LIN {X 0,Y 229.65,Z 466.167,A -85,B 0,C 180,E1 -20819.777,E2 -20819.777} C_VEL
LIN {X 0,Y 225.789,Z 455.718,A -85,B 0,C 180,E1 -20821.607,E2 -20821.607} C_VEL
LIN {X 0,Y 220.787,Z 444.949,A -85,B 0,C 180,E1 -20823.43,E2 -20823.43} C_VEL
LIN {X 0,Y 215.475,Z 435.139,A -85,B 0,C 180,E1 -20825.063,E2 -20825.063} C_VEL
LIN {X 0,Y 214,Z 432.562,A -85,B 0,C 180,E1 -20825.471,E2 -20825.471} C_VEL
LIN {X 0,Y 213.743,Z 431.361,A -85,B 0,C 180,E1 -20825.592,E2 -20825.592} C_VEL
LIN {X 0,Y 213.779,Z 431.357,A -85,B 0,C 180,E1 -20828.655,E2 -20828.655} C_VEL
LIN {X 0,Y 213.791,Z 431.354,A -85,B 0,C 180,E1 -20831.107,E2 -20831.107} C_VEL
LIN {X 0,Y 213.806,Z 431.352,A -85,B 0,C 180,E1 -20833.686,E2 -20833.686} C_VEL
LIN {X 0,Y 213.727,Z 431.361,A -85,B 0,C 180,E1 -20838.88,E2 -20838.88} C_VEL
LIN {X 0,Y 213.75,Z 431.36,A -85,B 0,C 180,E1 -20843.714,E2 -20843.714} C_VEL
LIN {X 0,Y 213.794,Z 431.352,A -85,B 0,C 180,E1 -20848.725,E2 -20848.725} C_VEL
LIN {X 0,Y 213.824,Z 431.35,A -85,B 0,C 180,E1 -20852.604,E2 -20852.604} C_VEL
LIN {X 0,Y 213.85,Z 431.346,A -85,B 0,C 180,E1 -20856.954,E2 -20856.954} C_VEL
LIN {X 0,Y 213.942,Z 431.334,A -85,B 0,C 180,E1 -20862.805,E2 -20862.805} C_VEL
LIN {X 0,Y 213.979,Z 431.329,A -85,B 0,C 180,E1 -20866.709,E2 -20866.709} C_VEL
LIN {X 0,Y 214.166,Z 431.302,A -85,B 0,C 180,E1 -20870.557,E2 -20870.557} C_VEL
LIN {X 0,Y 214.226,Z 431.299,A -85,B 0,C 180,E1 -20872.461,E2 -20872.461} C_VEL
LIN {X 0,Y 214.445,Z 431.245,A -85,B 0,C 180,E1 -20878.123,E2 -20878.123} C_VEL
LIN {X 0,Y 214.549,Z 431.244,A -85,B 0,C 180,E1 -20880.001,E2 -20880.001} C_VEL
LIN {X 0,Y 214.445,Z 431.271,A -85,B 0,C 180,E1 -20881.879,E2 -20881.879} C_VEL
LIN {X 0,Y 214.248,Z 431.3,A -85,B 0,C 180,E1 -20887.541,E2 -20887.541} C_VEL
LIN {X 0,Y 214.042,Z 431.325,A -85,B 0,C 180,E1 -20891.363,E2 -20891.363} C_VEL
LIN {X 0,Y 213.934,Z 431.338,A -85,B 0,C 180,E1 -20895.238,E2 -20895.238} C_VEL
LIN {X 0,Y 213.841,Z 431.349,A -85,B 0,C 180,E1 -20899.188,E2 -20899.188} C_VEL
LIN {X 0,Y 213.848,Z 431.35,A -85,B 0,C 180,E1 -20903.228,E2 -20903.228} C_VEL
LIN {X 0,Y 213.864,Z 431.711,A -85,B 0,C 180,E1 -20907.393,E2 -20907.393} C_VEL
LIN {X 0,Y 214.059,Z 433.405,A -85,B 0,C 180,E1 -20911.691,E2 -20911.691} C_VEL
LIN {X 0,Y 214.301,Z 435.41,A -85,B 0,C 180,E1 -20916.18,E2 -20916.18} C_VEL
LIN {X 0,Y 214.681,Z 437.889,A -85,B 0,C 180,E1 -20921.154,E2 -20921.154} C_VEL
LIN {X 0,Y 214.855,Z 439.419,A -85,B 0,C 180,E1 -20923.976,E2 -20923.976} C_VEL
LIN {X 0,Y 214.881,Z 440.961,A -85,B 0,C 180,E1 -20926.62,E2 -20926.62} C_VEL
LIN {X 0,Y 214.731,Z 442.501,A -85,B 0,C 180,E1 -20929.112,E2 -20929.112} C_VEL
LIN {X 0,Y 213.923,Z 445.534,A -85,B 0,C 180,E1 -20933.747,E2 -20933.747} C_VEL
LIN {X 0,Y 213.756,Z 446.179,A -85,B 0,C 180,E1 -20934.654,E2 -20934.654} C_VEL
LIN {X 0,Y 214.719,Z 449.544,A -85,B 0,C 180,E1 -20935.029,E2 -20935.029} C_VEL
LIN {X 0,Y 218.657,Z 461.683,A -85,B 0,C 180,E1 -20936.689,E2 -20936.689} C_VEL
LIN {X 0,Y 221.392,Z 472.962,A -85,B 0,C 180,E1 -20938.374,E2 -20938.374} C_VEL
LIN {X 0,Y 222.956,Z 483.058,A -85,B 0,C 180,E1 -20939.999,E2 -20939.999} C_VEL
LIN {X 0,Y 223.803,Z 491.807,A -85,B 0,C 180,E1 -20941.557,E2 -20941.557} C_VEL
LIN {X 0,Y 223.936,Z 501.293,A -85,B 0,C 180,E1 -20943.435,E2 -20943.435} C_VEL
LIN {X 0,Y 223.732,Z 505.859,A -85,B 0,C 180,E1 -20944.41,E2 -20944.41} C_VEL
LIN {X 0,Y 220.785,Z 516.308,A -85,B 0,C 180,E1 -20946.818,E2 -20946.818} C_VEL
LIN {X 0,Y 219.001,Z 523.013,A -85,B 0,C 180,E1 -20948.742,E2 -20948.742} C_VEL
LIN {X 0,Y 216.849,Z 529.814,A -85,B 0,C 180,E1 -20951.089,E2 -20951.089} C_VEL
LIN {X 0,Y 215.381,Z 534.744,A -85,B 0,C 180,E1 -20953.138,E2 -20953.138} C_VEL
LIN {X 0,Y 213.858,Z 537.614,A -85,B 0,C 180,E1 -20954.475,E2 -20954.475} C_VEL
LIN {X 0,Y 209.85,Z 541.622,A -85,B 0,C 180,E1 -20956.666,E2 -20956.666} C_VEL
LIN {X 0,Y 206.092,Z 545.045,A -85,B 0,C 180,E1 -20959.012,E2 -20959.012} C_VEL
LIN {X 0,Y 204.987,Z 546.698,A -85,B 0,C 180,E1 -20960.564,E2 -20960.564} C_VEL
LIN {X 0,Y 204.442,Z 549.502,A -85,B 0,C 180,E1 -20964.08,E2 -20964.08} C_VEL
LIN {X 0,Y 204.339,Z 550.566,A -85,B 0,C 180,E1 -20966.055,E2 -20966.055} C_VEL
LIN {X 0,Y 204.365,Z 551.161,A -85,B 0,C 180,E1 -20968.029,E2 -20968.029} C_VEL
LIN {X 0,Y 204.429,Z 551.319,A -85,B 0,C 180,E1 -20970,E2 -20970} C_VEL
LIN {X 0,Y 204.365,Z 551.161,A -85,B 0,C 180,E1 -20971.97,E2 -20971.97} C_VEL
LIN {X 0,Y 204.36,Z 550.491,A -85,B 0,C 180,E1 -20974.184,E2 -20974.184} C_VEL
LIN {X 0,Y 204.675,Z 548.109,A -85,B 0,C 180,E1 -20977.894,E2 -20977.894} C_VEL
LIN {X 0,Y 205.363,Z 545.153,A -85,B 0,C 180,E1 -20980.849,E2 -20980.849} C_VEL
LIN {X 0,Y 206.414,Z 541.157,A -85,B 0,C 180,E1 -20983.788,E2 -20983.788} C_VEL
LIN {X 0,Y 208.046,Z 536.024,A -85,B 0,C 180,E1 -20986.686,E2 -20986.686} C_VEL
LIN {X 0,Y 209.722,Z 530.759,A -85,B 0,C 180,E1 -20989.07,E2 -20989.07} C_VEL
LIN {X 0,Y 211.844,Z 524.444,A -85,B 0,C 180,E1 -20991.402,E2 -20991.402} C_VEL
LIN {X 0,Y 213.537,Z 518.486,A -85,B 0,C 180,E1 -20993.262,E2 -20993.262} C_VEL
LIN {X 0,Y 215.597,Z 511.56,A -85,B 0,C 180,E1 -20995.072,E2 -20995.072} C_VEL
LIN {X 0,Y 217.256,Z 505.648,A -85,B 0,C 180,E1 -20996.409,E2 -20996.409} C_VEL
LIN {X 0,Y 217.344,Z 495.828,A -85,B 0,C 180,E1 -20998.546,E2 -20998.546} C_VEL
LIN {X 0,Y 216.761,Z 486.56,A -85,B 0,C 180,E1 -21000.341,E2 -21000.341} C_VEL
LIN {X 0,Y 215.486,Z 477.1,A -85,B 0,C 180,E1 -21002.006,E2 -21002.006} C_VEL
LIN {X 0,Y 213.303,Z 466.615,A -85,B 0,C 180,E1 -21003.699,E2 -21003.699} C_VEL
LIN {X 0,Y 210.591,Z 457.078,A -85,B 0,C 180,E1 -21005.148,E2 -21005.148} C_VEL
LIN {X 0,Y 207.683,Z 448.976,A -85,B 0,C 180,E1 -21006.358,E2 -21006.358} C_VEL
LIN {X 0,Y 206.901,Z 445.966,A -85,B 0,C 180,E1 -21006.726,E2 -21006.726} C_VEL
LIN {X 0,Y 207.477,Z 443.775,A -85,B 0,C 180,E1 -21010.059,E2 -21010.059} C_VEL
LIN {X 0,Y 207.749,Z 442.248,A -85,B 0,C 180,E1 -21012.576,E2 -21012.576} C_VEL
LIN {X 0,Y 207.813,Z 440.729,A -85,B 0,C 180,E1 -21015.25,E2 -21015.25} C_VEL
LIN {X 0,Y 207.522,Z 438.25,A -85,B 0,C 180,E1 -21019.948,E2 -21019.948} C_VEL
LIN {X 0,Y 207.228,Z 435.972,A -85,B 0,C 180,E1 -21024.791,E2 -21024.791} C_VEL
LIN {X 0,Y 206.982,Z 434.053,A -85,B 0,C 180,E1 -21029.38,E2 -21029.38} C_VEL
LIN {X 0,Y 206.751,Z 432.425,A -85,B 0,C 180,E1 -21033.774,E2 -21033.774} C_VEL
LIN {X 0,Y 206.756,Z 432.236,A -85,B 0,C 180,E1 -21038.042,E2 -21038.042} C_VEL
LIN {X 0,Y 206.871,Z 432.219,A -85,B 0,C 180,E1 -21042.195,E2 -21042.195} C_VEL
LIN {X 0,Y 206.893,Z 432.214,A -85,B 0,C 180,E1 -21046.243,E2 -21046.243} C_VEL
LIN {X 0,Y 207.13,Z 432.185,A -85,B 0,C 180,E1 -21050.231,E2 -21050.231} C_VEL
LIN {X 0,Y 207.185,Z 432.178,A -85,B 0,C 180,E1 -21052.201,E2 -21052.201} C_VEL
LIN {X 0,Y 207.379,Z 432.152,A -85,B 0,C 180,E1 -21058.057,E2 -21058.057} C_VEL
LIN {X 0,Y 207.511,Z 432.119,A -85,B 0,C 180,E1 -21059.999,E2 -21059.999} C_VEL
LIN {X 0,Y 207.378,Z 432.124,A -85,B 0,C 180,E1 -21061.941,E2 -21061.941} C_VEL
LIN {X 0,Y 207.164,Z 432.18,A -85,B 0,C 180,E1 -21067.798,E2 -21067.798} C_VEL
LIN {X 0,Y 206.977,Z 432.202,A -85,B 0,C 180,E1 -21071.754,E2 -21071.754} C_VEL
LIN {X 0,Y 206.862,Z 432.211,A -85,B 0,C 180,E1 -21075.77,E2 -21075.77} C_VEL
LIN {X 0,Y 206.779,Z 432.222,A -85,B 0,C 180,E1 -21079.868,E2 -21079.868} C_VEL
LIN {X 0,Y 206.758,Z 432.225,A -85,B 0,C 180,E1 -21084.071,E2 -21084.071} C_VEL
LIN {X 0,Y 206.739,Z 432.231,A -85,B 0,C 180,E1 -21088.418,E2 -21088.418} C_VEL
LIN {X 0,Y 206.704,Z 432.236,A -85,B 0,C 180,E1 -21092.955,E2 -21092.955} C_VEL
LIN {X 0,Y 206.721,Z 432.235,A -85,B 0,C 180,E1 -21097.73,E2 -21097.73} C_VEL
LIN {X 0,Y 206.744,Z 432.233,A -85,B 0,C 180,E1 -21101.596,E2 -21101.596} C_VEL
LIN {X 0,Y 206.741,Z 432.232,A -85,B 0,C 180,E1 -21105.55,E2 -21105.55} C_VEL
LIN {X 0,Y 206.739,Z 432.232,A -85,B 0,C 180,E1 -21109.768,E2 -21109.768} C_VEL
LIN {X 0,Y 206.711,Z 432.331,A -85,B 0,C 180,E1 -21113.059,E2 -21113.059} C_VEL
LIN {X 0,Y 207.683,Z 435.05,A -85,B 0,C 180,E1 -21113.417,E2 -21113.417} C_VEL
LIN {X 0,Y 209.172,Z 437.265,A -85,B 0,C 180,E1 -21113.847,E2 -21113.847} C_VEL
LIN {X 0,Y 214.507,Z 447.106,A -85,B 0,C 180,E1 -21115.615,E2 -21115.615} C_VEL
LIN {X 0,Y 218.684,Z 456.158,A -85,B 0,C 180,E1 -21117.262,E2 -21117.262} C_VEL
LIN {X 0,Y 222.353,Z 465.597,A -85,B 0,C 180,E1 -21119.035,E2 -21119.035} C_VEL
LIN {X 0,Y 225.766,Z 476.018,A -85,B 0,C 180,E1 -21121.121,E2 -21121.121} C_VEL
LIN {X 0,Y 229.479,Z 484.805,A -85,B 0,C 180,E1 -21123.22,E2 -21123.22} C_VEL
LIN {X 0,Y 234.862,Z 494.211,A -85,B 0,C 180,E1 -21125.874,E2 -21125.874} C_VEL
LIN {X 0,Y 241.471,Z 502.648,A -85,B 0,C 180,E1 -21128.645,E2 -21128.645} C_VEL
LIN {X 0,Y 249.05,Z 510.339,A -85,B 0,C 180,E1 -21131.527,E2 -21131.527} C_VEL
LIN {X 0,Y 256.368,Z 516.421,A -85,B 0,C 180,E1 -21134.09,E2 -21134.09} C_VEL
LIN {X 0,Y 263.767,Z 521.712,A -85,B 0,C 180,E1 -21136.585,E2 -21136.585} C_VEL
LIN {X 0,Y 270.068,Z 525.746,A -85,B 0,C 180,E1 -21138.71,E2 -21138.71} C_VEL
LIN {X 0,Y 277.243,Z 530.01,A -85,B 0,C 180,E1 -21141.347,E2 -21141.347} C_VEL
LIN {X 0,Y 280.836,Z 531.995,A -85,B 0,C 180,E1 -21142.812,E2 -21142.812} C_VEL
LIN {X 0,Y 283.81,Z 533.702,A -85,B 0,C 180,E1 -21144.316,E2 -21144.316} C_VEL
LIN {X 0,Y 285.973,Z 535.014,A -85,B 0,C 180,E1 -21145.772,E2 -21145.772} C_VEL
LIN {X 0,Y 288.419,Z 536.106,A -85,B 0,C 180,E1 -21147.495,E2 -21147.495} C_VEL
LIN {X 0,Y 289.599,Z 536.494,A -85,B 0,C 180,E1 -21148.61,E2 -21148.61} C_VEL
LIN {X 0,Y 290.596,Z 536.662,A -85,B 0,C 180,E1 -21150,E2 -21150} C_VEL
LIN {X 0,Y 289.595,Z 536.494,A -85,B 0,C 180,E1 -21151.391,E2 -21151.391} C_VEL
LIN {X 0,Y 287.975,Z 535.95,A -85,B 0,C 180,E1 -21152.798,E2 -21152.798} C_VEL
LIN {X 0,Y 285.954,Z 535.014,A -85,B 0,C 180,E1 -21154.229,E2 -21154.229} C_VEL
LIN {X 0,Y 282.8,Z 533.095,A -85,B 0,C 180,E1 -21156.257,E2 -21156.257} C_VEL
LIN {X 0,Y 280.804,Z 531.995,A -85,B 0,C 180,E1 -21157.189,E2 -21157.189} C_VEL
LIN {X 0,Y 274.892,Z 528.624,A -85,B 0,C 180,E1 -21159.566,E2 -21159.566} C_VEL
LIN {X 0,Y 267.715,Z 524.214,A -85,B 0,C 180,E1 -21162.123,E2 -21162.123} C_VEL
LIN {X 0,Y 258.513,Z 518.022,A -85,B 0,C 180,E1 -21165.186,E2 -21165.186} C_VEL
LIN {X 0,Y 250.424,Z 511.545,A -85,B 0,C 180,E1 -21167.981,E2 -21167.981} C_VEL
LIN {X 0,Y 242.862,Z 504.195,A -85,B 0,C 180,E1 -21170.799,E2 -21170.799} C_VEL
LIN {X 0,Y 235.936,Z 495.724,A -85,B 0,C 180,E1 -21173.66,E2 -21173.66} C_VEL
LIN {X 0,Y 230.601,Z 487.089,A -85,B 0,C 180,E1 -21176.18,E2 -21176.18} C_VEL
LIN {X 0,Y 226.199,Z 477.235,A -85,B 0,C 180,E1 -21178.617,E2 -21178.617} C_VEL
LIN {X 0,Y 222.351,Z 465.618,A -85,B 0,C 180,E1 -21180.963,E2 -21180.963} C_VEL
LIN {X 0,Y 219.408,Z 457.77,A -85,B 0,C 180,E1 -21182.441,E2 -21182.441} C_VEL
LIN {X 0,Y 214.209,Z 446.412,A -85,B 0,C 180,E1 -21184.497,E2 -21184.497} C_VEL
LIN {X 0,Y 208.574,Z 436.22,A -85,B 0,C 180,E1 -21186.355,E2 -21186.355} C_VEL
LIN {X 0,Y 207.02,Z 433.644,A -85,B 0,C 180,E1 -21186.817,E2 -21186.817} C_VEL
LIN {X 0,Y 206.702,Z 432.238,A -85,B 0,C 180,E1 -21187.013,E2 -21187.013} C_VEL
LIN {X 0,Y 206.721,Z 432.235,A -85,B 0,C 180,E1 -21191.589,E2 -21191.589} C_VEL
LIN {X 0,Y 206.671,Z 432.24,A -85,B 0,C 180,E1 -21195.571,E2 -21195.571} C_VEL
LIN {X 0,Y 206.67,Z 432.24,A -85,B 0,C 180,E1 -21199.753,E2 -21199.753} C_VEL
LIN {X 0,Y 206.729,Z 432.234,A -85,B 0,C 180,E1 -21204.696,E2 -21204.696} C_VEL
LIN {X 0,Y 206.721,Z 432.233,A -85,B 0,C 180,E1 -21209.34,E2 -21209.34} C_VEL
LIN {X 0,Y 206.73,Z 432.231,A -85,B 0,C 180,E1 -21213.773,E2 -21213.773} C_VEL
LIN {X 0,Y 206.756,Z 432.23,A -85,B 0,C 180,E1 -21218.044,E2 -21218.044} C_VEL
LIN {X 0,Y 206.872,Z 432.217,A -85,B 0,C 180,E1 -21222.198,E2 -21222.198} C_VEL
LIN {X 0,Y 206.912,Z 432.209,A -85,B 0,C 180,E1 -21226.247,E2 -21226.247} C_VEL
LIN {X 0,Y 207.104,Z 432.181,A -85,B 0,C 180,E1 -21230.232,E2 -21230.232} C_VEL
LIN {X 0,Y 207.167,Z 432.18,A -85,B 0,C 180,E1 -21232.202,E2 -21232.202} C_VEL
LIN {X 0,Y 207.381,Z 432.123,A -85,B 0,C 180,E1 -21238.059,E2 -21238.059} C_VEL
LIN {X 0,Y 207.514,Z 432.119,A -85,B 0,C 180,E1 -21240.001,E2 -21240.001} C_VEL
LIN {X 0,Y 207.382,Z 432.151,A -85,B 0,C 180,E1 -21241.943,E2 -21241.943} C_VEL
LIN {X 0,Y 207.188,Z 432.178,A -85,B 0,C 180,E1 -21247.799,E2 -21247.799} C_VEL
LIN {X 0,Y 206.975,Z 432.205,A -85,B 0,C 180,E1 -21251.757,E2 -21251.757} C_VEL
LIN {X 0,Y 206.867,Z 432.217,A -85,B 0,C 180,E1 -21255.772,E2 -21255.772} C_VEL
LIN {X 0,Y 206.785,Z 432.228,A -85,B 0,C 180,E1 -21259.87,E2 -21259.87} C_VEL
LIN {X 0,Y 206.765,Z 432.231,A -85,B 0,C 180,E1 -21264.073,E2 -21264.073} C_VEL
LIN {X 0,Y 206.753,Z 432.419,A -85,B 0,C 180,E1 -21266.226,E2 -21266.226} C_VEL
LIN {X 0,Y 206.983,Z 434.052,A -85,B 0,C 180,E1 -21270.62,E2 -21270.62} C_VEL
LIN {X 0,Y 207.24,Z 436.124,A -85,B 0,C 180,E1 -21275.522,E2 -21275.522} C_VEL
LIN {X 0,Y 207.532,Z 438.281,A -85,B 0,C 180,E1 -21280.049,E2 -21280.049} C_VEL
LIN {X 0,Y 207.816,Z 440.733,A -85,B 0,C 180,E1 -21284.75,E2 -21284.75} C_VEL
LIN {X 0,Y 207.713,Z 442.682,A -85,B 0,C 180,E1 -21288.107,E2 -21288.107} C_VEL
LIN {X 0,Y 207.079,Z 445.313,A -85,B 0,C 180,E1 -21292.346,E2 -21292.346} C_VEL
LIN {X 0,Y 206.918,Z 445.942,A -85,B 0,C 180,E1 -21293.271,E2 -21293.271} C_VEL
LIN {X 0,Y 207.954,Z 449.448,A -85,B 0,C 180,E1 -21293.724,E2 -21293.724} C_VEL
LIN {X 0,Y 211.693,Z 460.424,A -85,B 0,C 180,E1 -21295.339,E2 -21295.339} C_VEL
LIN {X 0,Y 214.495,Z 471.91,A -85,B 0,C 180,E1 -21297.121,E2 -21297.121} C_VEL
LIN {X 0,Y 216.225,Z 481.921,A -85,B 0,C 180,E1 -21298.814,E2 -21298.814} C_VEL
LIN {X 0,Y 217.133,Z 491.348,A -85,B 0,C 180,E1 -21300.553,E2 -21300.553} C_VEL
LIN {X 0,Y 217.336,Z 500.293,A -85,B 0,C 180,E1 -21302.384,E2 -21302.384} C_VEL
LIN {X 0,Y 217.035,Z 506.736,A -85,B 0,C 180,E1 -21303.819,E2 -21303.819} C_VEL
LIN {X 0,Y 214.528,Z 515.228,A -85,B 0,C 180,E1 -21305.826,E2 -21305.826} C_VEL
LIN {X 0,Y 212.183,Z 523.398,A -85,B 0,C 180,E1 -21308.246,E2 -21308.246} C_VEL
LIN {X 0,Y 210.126,Z 529.602,A -85,B 0,C 180,E1 -21310.46,E2 -21310.46} C_VEL
LIN {X 0,Y 208.451,Z 534.886,A -85,B 0,C 180,E1 -21312.747,E2 -21312.747} C_VEL
LIN {X 0,Y 206.897,Z 539.6,A -85,B 0,C 180,E1 -21315.24,E2 -21315.24} C_VEL
LIN {X 0,Y 205.685,Z 543.933,A -85,B 0,C 180,E1 -21318.17,E2 -21318.17} C_VEL
LIN {X 0,Y 204.987,Z 546.698,A -85,B 0,C 180,E1 -21320.564,E2 -21320.564} C_VEL
LIN {X 0,Y 203.992,Z 548.181,A -85,B 0,C 180,E1 -21322.151,E2 -21322.151} C_VEL
LIN {X 0,Y 200.828,Z 549.866,A -85,B 0,C 180,E1 -21324.77,E2 -21324.77} C_VEL
LIN {X 0,Y 198.342,Z 550.682,A -85,B 0,C 180,E1 -21326.935,E2 -21326.935} C_VEL
LIN {X 0,Y 197.287,Z 551.105,A -85,B 0,C 180,E1 -21328.918,E2 -21328.918} C_VEL
LIN {X 0,Y 197.278,Z 551.046,A -85,B 0,C 180,E1 -21329.206,E2 -21329.206} C_VEL
LIN {X 0,Y 197.271,Z 550.95,A -85,B 0,C 180,E1 -21332.041,E2 -21332.041} C_VEL
LIN {X 0,Y 197.257,Z 550.355,A -85,B 0,C 180,E1 -21334.086,E2 -21334.086} C_VEL
LIN {X 0,Y 197.642,Z 547.898,A -85,B 0,C 180,E1 -21338.177,E2 -21338.177} C_VEL
LIN {X 0,Y 198.355,Z 544.94,A -85,B 0,C 180,E1 -21341.237,E2 -21341.237} C_VEL
LIN {X 0,Y 199.484,Z 540.944,A -85,B 0,C 180,E1 -21344.277,E2 -21344.277} C_VEL
LIN {X 0,Y 201.227,Z 535.812,A -85,B 0,C 180,E1 -21347.269,E2 -21347.269} C_VEL
LIN {X 0,Y 202.996,Z 530.547,A -85,B 0,C 180,E1 -21349.727,E2 -21349.727} C_VEL
LIN {X 0,Y 205.216,Z 524.231,A -85,B 0,C 180,E1 -21352.13,E2 -21352.13} C_VEL
LIN {X 0,Y 207.005,Z 518.274,A -85,B 0,C 180,E1 -21354.041,E2 -21354.041} C_VEL
LIN {X 0,Y 209.157,Z 511.347,A -85,B 0,C 180,E1 -21355.9,E2 -21355.9} C_VEL
LIN {X 0,Y 210.587,Z 506.525,A -85,B 0,C 180,E1 -21357.046,E2 -21357.046} C_VEL
LIN {X 0,Y 210.738,Z 495.603,A -85,B 0,C 180,E1 -21359.528,E2 -21359.528} C_VEL
LIN {X 0,Y 210.24,Z 487.03,A -85,B 0,C 180,E1 -21361.268,E2 -21361.268} C_VEL
LIN {X 0,Y 208.916,Z 477.245,A -85,B 0,C 180,E1 -21363.086,E2 -21363.086} C_VEL
LIN {X 0,Y 206.806,Z 467.121,A -85,B 0,C 180,E1 -21364.823,E2 -21364.823} C_VEL
LIN {X 0,Y 203.968,Z 457.172,A -85,B 0,C 180,E1 -21366.44,E2 -21366.44} C_VEL
LIN {X 0,Y 201.106,Z 449.237,A -85,B 0,C 180,E1 -21367.719,E2 -21367.719} C_VEL
LIN {X 0,Y 200.134,Z 446.251,A -85,B 0,C 180,E1 -21368.111,E2 -21368.111} C_VEL
LIN {X 0,Y 200.126,Z 445.72,A -85,B 0,C 180,E1 -21368.233,E2 -21368.233} C_VEL
LIN {X 0,Y 200.695,Z 443.02,A -85,B 0,C 180,E1 -21372.659,E2 -21372.659} C_VEL
LIN {X 0,Y 200.731,Z 441.423,A -85,B 0,C 180,E1 -21375.552,E2 -21375.552} C_VEL
LIN {X 0,Y 200.613,Z 440.026,A -85,B 0,C 180,E1 -21378.269,E2 -21378.269} C_VEL
LIN {X 0,Y 200.232,Z 437.619,A -85,B 0,C 180,E1 -21383.366,E2 -21383.366} C_VEL
LIN {X 0,Y 200.005,Z 435.585,A -85,B 0,C 180,E1 -21388.19,E2 -21388.19} C_VEL
LIN {X 0,Y 199.782,Z 433.885,A -85,B 0,C 180,E1 -21392.785,E2 -21392.785} C_VEL
LIN {X 0,Y 199.679,Z 433.141,A -85,B 0,C 180,E1 -21395.015,E2 -21395.015} C_VEL
LIN {X 0,Y 199.698,Z 433.115,A -85,B 0,C 180,E1 -21399.393,E2 -21399.393} C_VEL
LIN {X 0,Y 199.802,Z 433.097,A -85,B 0,C 180,E1 -21403.655,E2 -21403.655} C_VEL
LIN {X 0,Y 200.066,Z 433.064,A -85,B 0,C 180,E1 -21409.601,E2 -21409.601} C_VEL
LIN {X 0,Y 200.129,Z 433.056,A -85,B 0,C 180,E1 -21411.924,E2 -21411.924} C_VEL
LIN {X 0,Y 200.319,Z 433.031,A -85,B 0,C 180,E1 -21417.988,E2 -21417.988} C_VEL
LIN {X 0,Y 200.476,Z 432.995,A -85,B 0,C 180,E1 -21419.999,E2 -21419.999} C_VEL
LIN {X 0,Y 200.027,Z 433.052,A -85,B 0,C 180,E1 -21424.028,E2 -21424.028} C_VEL
LIN {X 0,Y 200.107,Z 433.058,A -85,B 0,C 180,E1 -21428.075,E2 -21428.075} C_VEL
LIN {X 0,Y 199.909,Z 433.085,A -85,B 0,C 180,E1 -21432.176,E2 -21432.176} C_VEL
LIN {X 0,Y 199.8,Z 433.095,A -85,B 0,C 180,E1 -21436.343,E2 -21436.343} C_VEL
LIN {X 0,Y 199.695,Z 433.105,A -85,B 0,C 180,E1 -21440.605,E2 -21440.605} C_VEL
LIN {X 0,Y 199.668,Z 433.105,A -85,B 0,C 180,E1 -21444.984,E2 -21444.984} C_VEL
LIN {X 0,Y 199.67,Z 433.113,A -85,B 0,C 180,E1 -21449.522,E2 -21449.522} C_VEL
LIN {X 0,Y 199.659,Z 433.115,A -85,B 0,C 180,E1 -21452.352,E2 -21452.352} C_VEL
LIN {X 0,Y 199.649,Z 433.116,A -85,B 0,C 180,E1 -21456.756,E2 -21456.756} C_VEL
LIN {X 0,Y 199.697,Z 433.11,A -85,B 0,C 180,E1 -21459.306,E2 -21459.306} C_VEL
LIN {X 0,Y 199.685,Z 433.11,A -85,B 0,C 180,E1 -21462.346,E2 -21462.346} C_VEL
LIN {X 0,Y 199.689,Z 433.11,A -85,B 0,C 180,E1 -21465.261,E2 -21465.261} C_VEL
LIN {X 0,Y 199.689,Z 433.112,A -85,B 0,C 180,E1 -21468.035,E2 -21468.035} C_VEL
LIN {X 0,Y 199.714,Z 433.109,A -85,B 0,C 180,E1 -21471.537,E2 -21471.537} C_VEL
LIN {X 0,Y 200.699,Z 435.981,A -85,B 0,C 180,E1 -21471.963,E2 -21471.963} C_VEL
LIN {X 0,Y 202.287,Z 438.351,A -85,B 0,C 180,E1 -21472.458,E2 -21472.458} C_VEL
LIN {X 0,Y 208.22,Z 449.114,A -85,B 0,C 180,E1 -21474.576,E2 -21474.576} C_VEL
LIN {X 0,Y 213.622,Z 461.247,A -85,B 0,C 180,E1 -21476.968,E2 -21476.968} C_VEL
LIN {X 0,Y 217.172,Z 471.377,A -85,B 0,C 180,E1 -21479.042,E2 -21479.042} C_VEL
LIN {X 0,Y 220.136,Z 480.806,A -85,B 0,C 180,E1 -21481.144,E2 -21481.144} C_VEL
LIN {X 0,Y 223.412,Z 488.445,A -85,B 0,C 180,E1 -21483.145,E2 -21483.145} C_VEL
LIN {X 0,Y 228.407,Z 497.265,A -85,B 0,C 180,E1 -21485.835,E2 -21485.835} C_VEL
LIN {X 0,Y 234.202,Z 504.732,A -85,B 0,C 180,E1 -21488.472,E2 -21488.472} C_VEL
LIN {X 0,Y 242.377,Z 512.893,A -85,B 0,C 180,E1 -21491.757,E2 -21491.757} C_VEL
LIN {X 0,Y 250.669,Z 519.436,A -85,B 0,C 180,E1 -21494.769,E2 -21494.769} C_VEL
LIN {X 0,Y 259.007,Z 524.859,A -85,B 0,C 180,E1 -21497.64,E2 -21497.64} C_VEL
LIN {X 0,Y 266.448,Z 529.095,A -85,B 0,C 180,E1 -21500.253,E2 -21500.253} C_VEL
LIN {X 0,Y 272.477,Z 532.246,A -85,B 0,C 180,E1 -21502.591,E2 -21502.591} C_VEL
LIN {X 0,Y 276.052,Z 533.935,A -85,B 0,C 180,E1 -21504.155,E2 -21504.155} C_VEL
LIN {X 0,Y 278.425,Z 535.238,A -85,B 0,C 180,E1 -21505.657,E2 -21505.657} C_VEL
LIN {X 0,Y 281.343,Z 536.422,A -85,B 0,C 180,E1 -21507.696,E2 -21507.696} C_VEL
LIN {X 0,Y 282.31,Z 536.71,A -85,B 0,C 180,E1 -21508.574,E2 -21508.574} C_VEL
LIN {X 0,Y 283.431,Z 536.871,A -85,B 0,C 180,E1 -21510,E2 -21510} C_VEL
LIN {X 0,Y 282.301,Z 536.71,A -85,B 0,C 180,E1 -21511.427,E2 -21511.427} C_VEL
LIN {X 0,Y 280.5,Z 536.174,A -85,B 0,C 180,E1 -21512.873,E2 -21512.873} C_VEL
LIN {X 0,Y 278.397,Z 535.238,A -85,B 0,C 180,E1 -21514.344,E2 -21514.344} C_VEL
LIN {X 0,Y 275.616,Z 533.754,A -85,B 0,C 180,E1 -21516.038,E2 -21516.038} C_VEL
LIN {X 0,Y 269.973,Z 530.945,A -85,B 0,C 180,E1 -21518.425,E2 -21518.425} C_VEL
LIN {X 0,Y 263.701,Z 527.524,A -85,B 0,C 180,E1 -21520.752,E2 -21520.752} C_VEL
LIN {X 0,Y 256.044,Z 523.008,A -85,B 0,C 180,E1 -21523.374,E2 -21523.374} C_VEL
LIN {X 0,Y 247.027,Z 516.707,A -85,B 0,C 180,E1 -21526.529,E2 -21526.529} C_VEL
LIN {X 0,Y 238.792,Z 509.57,A -85,B 0,C 180,E1 -21529.646,E2 -21529.646} C_VEL
LIN {X 0,Y 230.913,Z 500.773,A -85,B 0,C 180,E1 -21532.98,E2 -21532.98} C_VEL
LIN {X 0,Y 225.824,Z 493.03,A -85,B 0,C 180,E1 -21535.511,E2 -21535.511} C_VEL
LIN {X 0,Y 222.089,Z 485.673,A -85,B 0,C 180,E1 -21537.62,E2 -21537.62} C_VEL
LIN {X 0,Y 218.717,Z 476.723,A -85,B 0,C 180,E1 -21539.823,E2 -21539.823} C_VEL
LIN {X 0,Y 215.492,Z 466.218,A -85,B 0,C 180,E1 -21542.012,E2 -21542.012} C_VEL
LIN {X 0,Y 211.715,Z 456.784,A -85,B 0,C 180,E1 -21543.915,E2 -21543.915} C_VEL
LIN {X 0,Y 207.27,Z 447.354,A -85,B 0,C 180,E1 -21545.765,E2 -21545.765} C_VEL
LIN {X 0,Y 203.113,Z 439.932,A -85,B 0,C 180,E1 -21547.268,E2 -21547.268} C_VEL
LIN {X 0,Y 201.501,Z 437.039,A -85,B 0,C 180,E1 -21547.814,E2 -21547.814} C_VEL
LIN {X 0,Y 200.029,Z 434.483,A -85,B 0,C 180,E1 -21548.3,E2 -21548.3} C_VEL
LIN {X 0,Y 199.721,Z 433.108,A -85,B 0,C 180,E1 -21548.526,E2 -21548.526} C_VEL
LIN {X 0,Y 199.66,Z 433.114,A -85,B 0,C 180,E1 -21552.339,E2 -21552.339} C_VEL
LIN {X 0,Y 199.628,Z 433.117,A -85,B 0,C 180,E1 -21555.244,E2 -21555.244} C_VEL
LIN {X 0,Y 199.639,Z 433.117,A -85,B 0,C 180,E1 -21560.757,E2 -21560.757} C_VEL
LIN {X 0,Y 199.633,Z 433.119,A -85,B 0,C 180,E1 -21565.719,E2 -21565.719} C_VEL
LIN {X 0,Y 199.702,Z 433.109,A -85,B 0,C 180,E1 -21568.139,E2 -21568.139} C_VEL
LIN {X 0,Y 199.685,Z 433.111,A -85,B 0,C 180,E1 -21572.773,E2 -21572.773} C_VEL
LIN {X 0,Y 199.736,Z 433.104,A -85,B 0,C 180,E1 -21577.23,E2 -21577.23} C_VEL
LIN {X 0,Y 199.795,Z 433.096,A -85,B 0,C 180,E1 -21581.759,E2 -21581.759} C_VEL
LIN {X 0,Y 199.846,Z 433.085,A -85,B 0,C 180,E1 -21585.75,E2 -21585.75} C_VEL
LIN {X 0,Y 200.069,Z 433.057,A -85,B 0,C 180,E1 -21589.885,E2 -21589.885} C_VEL
LIN {X 0,Y 200.034,Z 433.065,A -85,B 0,C 180,E1 -21593.951,E2 -21593.951} C_VEL
LIN {X 0,Y 200.321,Z 433.001,A -85,B 0,C 180,E1 -21597.991,E2 -21597.991} C_VEL
LIN {X 0,Y 200.479,Z 432.994,A -85,B 0,C 180,E1 -21600.001,E2 -21600.001} C_VEL
LIN {X 0,Y 200.032,Z 433.067,A -85,B 0,C 180,E1 -21604.031,E2 -21604.031} C_VEL
LIN {X 0,Y 200.132,Z 433.056,A -85,B 0,C 180,E1 -21608.076,E2 -21608.076} C_VEL
LIN {X 0,Y 199.906,Z 433.084,A -85,B 0,C 180,E1 -21612.178,E2 -21612.178} C_VEL
LIN {X 0,Y 199.805,Z 433.096,A -85,B 0,C 180,E1 -21616.345,E2 -21616.345} C_VEL
LIN {X 0,Y 199.701,Z 433.11,A -85,B 0,C 180,E1 -21620.606,E2 -21620.606} C_VEL
LIN {X 0,Y 199.681,Z 433.134,A -85,B 0,C 180,E1 -21624.984,E2 -21624.984} C_VEL
LIN {X 0,Y 199.893,Z 434.686,A -85,B 0,C 180,E1 -21629.488,E2 -21629.488} C_VEL
LIN {X 0,Y 200.114,Z 436.562,A -85,B 0,C 180,E1 -21634.19,E2 -21634.19} C_VEL
LIN {X 0,Y 200.45,Z 438.961,A -85,B 0,C 180,E1 -21639.526,E2 -21639.526} C_VEL
LIN {X 0,Y 200.661,Z 440.503,A -85,B 0,C 180,E1 -21642.65,E2 -21642.65} C_VEL
LIN {X 0,Y 200.747,Z 442.036,A -85,B 0,C 180,E1 -21645.558,E2 -21645.558} C_VEL
LIN {X 0,Y 200.614,Z 443.565,A -85,B 0,C 180,E1 -21648.271,E2 -21648.271} C_VEL
LIN {X 0,Y 200.114,Z 445.744,A -85,B 0,C 180,E1 -21651.84,E2 -21651.84} C_VEL
LIN {X 0,Y 200.983,Z 448.988,A -85,B 0,C 180,E1 -21652.239,E2 -21652.239} C_VEL
LIN {X 0,Y 201.871,Z 451.031,A -85,B 0,C 180,E1 -21652.58,E2 -21652.58} C_VEL
LIN {X 0,Y 205.759,Z 463.012,A -85,B 0,C 180,E1 -21654.503,E2 -21654.503} C_VEL
LIN {X 0,Y 208.181,Z 473.356,A -85,B 0,C 180,E1 -21656.23,E2 -21656.23} C_VEL
LIN {X 0,Y 209.781,Z 482.876,A -85,B 0,C 180,E1 -21657.946,E2 -21657.946} C_VEL
LIN {X 0,Y 210.602,Z 492.033,A -85,B 0,C 180,E1 -21659.73,E2 -21659.73} C_VEL
LIN {X 0,Y 210.747,Z 499.548,A -85,B 0,C 180,E1 -21661.319,E2 -21661.319} C_VEL
LIN {X 0,Y 210.377,Z 507.507,A -85,B 0,C 180,E1 -21663.193,E2 -21663.193} C_VEL
LIN {X 0,Y 207.509,Z 516.643,A -85,B 0,C 180,E1 -21665.488,E2 -21665.488} C_VEL
LIN {X 0,Y 205.665,Z 522.661,A -85,B 0,C 180,E1 -21667.319,E2 -21667.319} C_VEL
LIN {X 0,Y 203.438,Z 529.39,A -85,B 0,C 180,E1 -21669.79,E2 -21669.79} C_VEL
LIN {X 0,Y 201.959,Z 533.895,A -85,B 0,C 180,E1 -21671.748,E2 -21671.748} C_VEL
LIN {X 0,Y 200.022,Z 539.388,A -85,B 0,C 180,E1 -21674.721,E2 -21674.721} C_VEL
LIN {X 0,Y 198.698,Z 543.72,A -85,B 0,C 180,E1 -21677.747,E2 -21677.747} C_VEL
LIN {X 0,Y 197.907,Z 546.669,A -85,B 0,C 180,E1 -21680.432,E2 -21680.432} C_VEL
LIN {X 0,Y 197.37,Z 549.29,A -85,B 0,C 180,E1 -21683.867,E2 -21683.867} C_VEL
LIN {X 0,Y 197.247,Z 550.406,A -85,B 0,C 180,E1 -21686.088,E2 -21686.088} C_VEL
LIN {X 0,Y 197.278,Z 551.046,A -85,B 0,C 180,E1 -21689.206,E2 -21689.206} C_VEL
LIN {X 0,Y 196.642,Z 551.109,A -85,B 0,C 180,E1 -21690.908,E2 -21690.908} C_VEL
LIN {X 0,Y 195.047,Z 550.788,A -85,B 0,C 180,E1 -21692.579,E2 -21692.579} C_VEL
LIN {X 0,Y 191.39,Z 549.327,A -85,B 0,C 180,E1 -21695.945,E2 -21695.945} C_VEL
LIN {X 0,Y 190.515,Z 548.104,A -85,B 0,C 180,E1 -21697.986,E2 -21697.986} C_VEL
LIN {X 0,Y 190.545,Z 547.817,A -85,B 0,C 180,E1 -21698.281,E2 -21698.281} C_VEL
LIN {X 0,Y 191.362,Z 544.728,A -85,B 0,C 180,E1 -21701.653,E2 -21701.653} C_VEL
LIN {X 0,Y 192.575,Z 540.732,A -85,B 0,C 180,E1 -21704.8,E2 -21704.8} C_VEL
LIN {X 0,Y 194.435,Z 535.6,A -85,B 0,C 180,E1 -21707.892,E2 -21707.892} C_VEL
LIN {X 0,Y 196.311,Z 530.335,A -85,B 0,C 180,E1 -21710.429,E2 -21710.429} C_VEL
LIN {X 0,Y 198.163,Z 525.396,A -85,B 0,C 180,E1 -21712.411,E2 -21712.411} C_VEL
LIN {X 0,Y 200.519,Z 518.062,A -85,B 0,C 180,E1 -21714.871,E2 -21714.871} C_VEL
LIN {X 0,Y 202.762,Z 511.135,A -85,B 0,C 180,E1 -21716.781,E2 -21716.781} C_VEL
LIN {X 0,Y 204.015,Z 506.304,A -85,B 0,C 180,E1 -21717.992,E2 -21717.992} C_VEL
LIN {X 0,Y 204.224,Z 496.693,A -85,B 0,C 180,E1 -21720.293,E2 -21720.293} C_VEL
LIN {X 0,Y 203.62,Z 486.425,A -85,B 0,C 180,E1 -21722.473,E2 -21722.473} C_VEL
LIN {X 0,Y 202.254,Z 476.419,A -85,B 0,C 180,E1 -21724.411,E2 -21724.411} C_VEL
LIN {X 0,Y 200.198,Z 466.843,A -85,B 0,C 180,E1 -21726.154,E2 -21726.154} C_VEL
LIN {X 0,Y 197.263,Z 456.978,A -85,B 0,C 180,E1 -21727.886,E2 -21727.886} C_VEL
LIN {X 0,Y 194.595,Z 449.459,A -85,B 0,C 180,E1 -21729.185,E2 -21729.185} C_VEL
LIN {X 0,Y 193.4,Z 446.347,A -85,B 0,C 180,E1 -21729.671,E2 -21729.671} C_VEL
LIN {X 0,Y 193.291,Z 445.528,A -85,B 0,C 180,E1 -21729.793,E2 -21729.793} C_VEL
LIN {X 0,Y 193.653,Z 443.323,A -85,B 0,C 180,E1 -21733.592,E2 -21733.592} C_VEL
LIN {X 0,Y 193.636,Z 441.769,A -85,B 0,C 180,E1 -21736.542,E2 -21736.542} C_VEL
LIN {X 0,Y 193.444,Z 440.246,A -85,B 0,C 180,E1 -21739.723,E2 -21739.723} C_VEL
LIN {X 0,Y 193.141,Z 438.184,A -85,B 0,C 180,E1 -21744.393,E2 -21744.393} C_VEL
LIN {X 0,Y 193.055,Z 437.155,A -85,B 0,C 180,E1 -21746.901,E2 -21746.901} C_VEL
LIN {X 0,Y 192.837,Z 435.348,A -85,B 0,C 180,E1 -21751.718,E2 -21751.718} C_VEL
LIN {X 0,Y 192.704,Z 433.988,A -85,B 0,C 180,E1 -21756.347,E2 -21756.347} C_VEL
LIN {X 0,Y 192.73,Z 433.98,A -85,B 0,C 180,E1 -21761.456,E2 -21761.456} C_VEL
LIN {X 0,Y 192.762,Z 433.974,A -85,B 0,C 180,E1 -21765.212,E2 -21765.212} C_VEL
LIN {X 0,Y 193.018,Z 433.942,A -85,B 0,C 180,E1 -21769.509,E2 -21769.509} C_VEL
LIN {X 0,Y 193.002,Z 433.944,A -85,B 0,C 180,E1 -21773.727,E2 -21773.727} C_VEL
LIN {X 0,Y 193.261,Z 433.911,A -85,B 0,C 180,E1 -21777.915,E2 -21777.915} C_VEL
LIN {X 0,Y 193.44,Z 433.87,A -85,B 0,C 180,E1 -21779.999,E2 -21779.999} C_VEL
LIN {X 0,Y 192.973,Z 433.93,A -85,B 0,C 180,E1 -21784.176,E2 -21784.176} C_VEL
LIN {X 0,Y 193.058,Z 433.934,A -85,B 0,C 180,E1 -21788.372,E2 -21788.372} C_VEL
LIN {X 0,Y 192.848,Z 433.963,A -85,B 0,C 180,E1 -21792.629,E2 -21792.629} C_VEL
LIN {X 0,Y 192.753,Z 433.974,A -85,B 0,C 180,E1 -21796.958,E2 -21796.958} C_VEL
LIN {X 0,Y 192.632,Z 433.987,A -85,B 0,C 180,E1 -21801.396,E2 -21801.396} C_VEL
LIN {X 0,Y 192.659,Z 433.98,A -85,B 0,C 180,E1 -21804.224,E2 -21804.224} C_VEL
LIN {X 0,Y 192.645,Z 433.986,A -85,B 0,C 180,E1 -21808.891,E2 -21808.891} C_VEL
LIN {X 0,Y 192.596,Z 433.994,A -85,B 0,C 180,E1 -21813.185,E2 -21813.185} C_VEL
LIN {X 0,Y 192.608,Z 433.992,A -85,B 0,C 180,E1 -21818.337,E2 -21818.337} C_VEL
LIN {X 0,Y 192.623,Z 433.989,A -85,B 0,C 180,E1 -21823.139,E2 -21823.139} C_VEL
LIN {X 0,Y 192.623,Z 433.991,A -85,B 0,C 180,E1 -21826.861,E2 -21826.861} C_VEL
LIN {X 0,Y 192.613,Z 433.992,A -85,B 0,C 180,E1 -21829.858,E2 -21829.858} C_VEL
LIN {X 0,Y 193.709,Z 436.944,A -85,B 0,C 180,E1 -21830.371,E2 -21830.371} C_VEL
LIN {X 0,Y 195.28,Z 439.033,A -85,B 0,C 180,E1 -21830.887,E2 -21830.887} C_VEL
LIN {X 0,Y 202.225,Z 451.797,A -85,B 0,C 180,E1 -21833.617,E2 -21833.617} C_VEL
LIN {X 0,Y 207.063,Z 462.813,A -85,B 0,C 180,E1 -21835.977,E2 -21835.977} C_VEL
LIN {X 0,Y 210.261,Z 471.751,A -85,B 0,C 180,E1 -21837.93,E2 -21837.93} C_VEL
LIN {X 0,Y 213.348,Z 482.276,A -85,B 0,C 180,E1 -21840.389,E2 -21840.389} C_VEL
LIN {X 0,Y 216.517,Z 490.489,A -85,B 0,C 180,E1 -21842.644,E2 -21842.644} C_VEL
LIN {X 0,Y 220.913,Z 498.698,A -85,B 0,C 180,E1 -21845.278,E2 -21845.278} C_VEL
LIN {X 0,Y 226.654,Z 506.433,A -85,B 0,C 180,E1 -21848.156,E2 -21848.156} C_VEL
LIN {X 0,Y 233.778,Z 513.725,A -85,B 0,C 180,E1 -21851.252,E2 -21851.252} C_VEL
LIN {X 0,Y 243.4,Z 521.216,A -85,B 0,C 180,E1 -21854.938,E2 -21854.938} C_VEL
LIN {X 0,Y 251.606,Z 526.274,A -85,B 0,C 180,E1 -21857.856,E2 -21857.856} C_VEL
LIN {X 0,Y 259.527,Z 530.379,A -85,B 0,C 180,E1 -21860.65,E2 -21860.65} C_VEL
LIN {X 0,Y 264.016,Z 532.5,A -85,B 0,C 180,E1 -21862.352,E2 -21862.352} C_VEL
LIN {X 0,Y 268.426,Z 534.398,A -85,B 0,C 180,E1 -21864.217,E2 -21864.217} C_VEL
LIN {X 0,Y 270.766,Z 535.465,A -85,B 0,C 180,E1 -21865.534,E2 -21865.534} C_VEL
LIN {X 0,Y 274.27,Z 536.73,A -85,B 0,C 180,E1 -21867.909,E2 -21867.909} C_VEL
LIN {X 0,Y 275.009,Z 536.926,A -85,B 0,C 180,E1 -21868.536,E2 -21868.536} C_VEL
LIN {X 0,Y 276.251,Z 537.081,A -85,B 0,C 180,E1 -21870,E2 -21870} C_VEL
LIN {X 0,Y 274.998,Z 536.926,A -85,B 0,C 180,E1 -21871.465,E2 -21871.465} C_VEL
LIN {X 0,Y 272.982,Z 536.4,A -85,B 0,C 180,E1 -21872.952,E2 -21872.952} C_VEL
LIN {X 0,Y 270.735,Z 535.465,A -85,B 0,C 180,E1 -21874.467,E2 -21874.467} C_VEL
LIN {X 0,Y 267.838,Z 534.181,A -85,B 0,C 180,E1 -21876.025,E2 -21876.025} C_VEL
LIN {X 0,Y 262.704,Z 531.865,A -85,B 0,C 180,E1 -21878.18,E2 -21878.18} C_VEL
LIN {X 0,Y 257.103,Z 529.147,A -85,B 0,C 180,E1 -21880.246,E2 -21880.246} C_VEL
LIN {X 0,Y 249.046,Z 524.787,A -85,B 0,C 180,E1 -21883.048,E2 -21883.048} C_VEL
LIN {X 0,Y 241.147,Z 519.602,A -85,B 0,C 180,E1 -21885.902,E2 -21885.902} C_VEL
LIN {X 0,Y 233.78,Z 513.72,A -85,B 0,C 180,E1 -21888.749,E2 -21888.749} C_VEL
LIN {X 0,Y 226.656,Z 506.43,A -85,B 0,C 180,E1 -21891.845,E2 -21891.845} C_VEL
LIN {X 0,Y 220.944,Z 498.671,A -85,B 0,C 180,E1 -21894.725,E2 -21894.725} C_VEL
LIN {X 0,Y 216.52,Z 490.466,A -85,B 0,C 180,E1 -21897.361,E2 -21897.361} C_VEL
LIN {X 0,Y 213.304,Z 482.273,A -85,B 0,C 180,E1 -21899.619,E2 -21899.619} C_VEL
LIN {X 0,Y 210.69,Z 473.287,A -85,B 0,C 180,E1 -21901.727,E2 -21901.727} C_VEL
LIN {X 0,Y 208.375,Z 466.192,A -85,B 0,C 180,E1 -21903.282,E2 -21903.282} C_VEL
LIN {X 0,Y 204.52,Z 456.839,A -85,B 0,C 180,E1 -21905.304,E2 -21905.304} C_VEL
LIN {X 0,Y 199.784,Z 447.192,A -85,B 0,C 180,E1 -21907.366,E2 -21907.366} C_VEL
LIN {X 0,Y 194.555,Z 438.01,A -85,B 0,C 180,E1 -21909.372,E2 -21909.372} C_VEL
LIN {X 0,Y 192.976,Z 435.546,A -85,B 0,C 180,E1 -21909.927,E2 -21909.927} C_VEL
LIN {X 0,Y 192.594,Z 433.994,A -85,B 0,C 180,E1 -21910.137,E2 -21910.137} C_VEL
LIN {X 0,Y 192.59,Z 433.996,A -85,B 0,C 180,E1 -21913.895,E2 -21913.895} C_VEL
LIN {X 0,Y 192.533,Z 434.001,A -85,B 0,C 180,E1 -21918.926,E2 -21918.926} C_VEL
LIN {X 0,Y 192.607,Z 433.993,A -85,B 0,C 180,E1 -21923.393,E2 -21923.393} C_VEL
LIN {X 0,Y 192.605,Z 433.993,A -85,B 0,C 180,E1 -21927.06,E2 -21927.06} C_VEL
LIN {X 0,Y 192.663,Z 433.985,A -85,B 0,C 180,E1 -21931.693,E2 -21931.693} C_VEL
LIN {X 0,Y 192.704,Z 433.979,A -85,B 0,C 180,E1 -21936.35,E2 -21936.35} C_VEL
LIN {X 0,Y 192.731,Z 433.975,A -85,B 0,C 180,E1 -21941.459,E2 -21941.459} C_VEL
LIN {X 0,Y 192.77,Z 433.965,A -85,B 0,C 180,E1 -21945.215,E2 -21945.215} C_VEL
LIN {X 0,Y 192.98,Z 433.941,A -85,B 0,C 180,E1 -21949.51,E2 -21949.51} C_VEL
LIN {X 0,Y 193.061,Z 433.933,A -85,B 0,C 180,E1 -21951.628,E2 -21951.628} C_VEL
LIN {X 0,Y 193.263,Z 433.879,A -85,B 0,C 180,E1 -21957.917,E2 -21957.917} C_VEL
LIN {X 0,Y 193.443,Z 433.869,A -85,B 0,C 180,E1 -21960.001,E2 -21960.001} C_VEL
LIN {X 0,Y 192.979,Z 433.946,A -85,B 0,C 180,E1 -21964.178,E2 -21964.178} C_VEL
LIN {X 0,Y 193.079,Z 433.934,A -85,B 0,C 180,E1 -21968.373,E2 -21968.373} C_VEL
LIN {X 0,Y 193.011,Z 433.943,A -85,B 0,C 180,E1 -21970.539,E2 -21970.539} C_VEL
LIN {X 0,Y 192.758,Z 433.975,A -85,B 0,C 180,E1 -21976.96,E2 -21976.96} C_VEL
LIN {X 0,Y 192.638,Z 433.992,A -85,B 0,C 180,E1 -21981.398,E2 -21981.398} C_VEL
LIN {X 0,Y 192.667,Z 434.016,A -85,B 0,C 180,E1 -21984.226,E2 -21984.226} C_VEL
LIN {X 0,Y 192.862,Z 435.604,A -85,B 0,C 180,E1 -21989.006,E2 -21989.006} C_VEL
LIN {X 0,Y 193.032,Z 437.172,A -85,B 0,C 180,E1 -21993.134,E2 -21993.134} C_VEL
LIN {X 0,Y 193.281,Z 439.296,A -85,B 0,C 180,E1 -21998.182,E2 -21998.182} C_VEL
LIN {X 0,Y 193.492,Z 440.527,A -85,B 0,C 180,E1 -22000.83,E2 -22000.83} C_VEL
LIN {X 0,Y 193.646,Z 441.885,A -85,B 0,C 180,E1 -22003.597,E2 -22003.597} C_VEL
LIN {X 0,Y 193.653,Z 443.412,A -85,B 0,C 180,E1 -22006.54,E2 -22006.54} C_VEL
LIN {X 0,Y 193.312,Z 445.555,A -85,B 0,C 180,E1 -22010.255,E2 -22010.255} C_VEL
LIN {X 0,Y 194.155,Z 448.603,A -85,B 0,C 180,E1 -22010.654,E2 -22010.654} C_VEL
LIN {X 0,Y 195.112,Z 450.74,A -85,B 0,C 180,E1 -22011.042,E2 -22011.042} C_VEL
LIN {X 0,Y 198.59,Z 460.818,A -85,B 0,C 180,E1 -22012.778,E2 -22012.778} C_VEL
LIN {X 0,Y 201.571,Z 472.882,A -85,B 0,C 180,E1 -22014.929,E2 -22014.929} C_VEL
LIN {X 0,Y 203.264,Z 483.008,A -85,B 0,C 180,E1 -22016.853,E2 -22016.853} C_VEL
LIN {X 0,Y 204.015,Z 491.947,A -85,B 0,C 180,E1 -22018.674,E2 -22018.674} C_VEL
LIN {X 0,Y 204.215,Z 499.863,A -85,B 0,C 180,E1 -22020.445,E2 -22020.445} C_VEL
LIN {X 0,Y 203.893,Z 507.29,A -85,B 0,C 180,E1 -22022.268,E2 -22022.268} C_VEL
LIN {X 0,Y 201.044,Z 516.431,A -85,B 0,C 180,E1 -22024.645,E2 -22024.645} C_VEL
LIN {X 0,Y 198.861,Z 523.116,A -85,B 0,C 180,E1 -22026.764,E2 -22026.764} C_VEL
LIN {X 0,Y 196.786,Z 529.179,A -85,B 0,C 180,E1 -22029.075,E2 -22029.075} C_VEL
LIN {X 0,Y 195.192,Z 533.683,A -85,B 0,C 180,E1 -22031.092,E2 -22031.092} C_VEL
LIN {X 0,Y 193.14,Z 539.176,A -85,B 0,C 180,E1 -22034.162,E2 -22034.162} C_VEL
LIN {X 0,Y 191.734,Z 543.508,A -85,B 0,C 180,E1 -22037.295,E2 -22037.295} C_VEL
LIN {X 0,Y 191.062,Z 545.88,A -85,B 0,C 180,E1 -22039.402,E2 -22039.402} C_VEL
LIN {X 0,Y 190.582,Z 547.685,A -85,B 0,C 180,E1 -22041.517,E2 -22041.517} C_VEL
LIN {X 0,Y 190.167,Z 550.143,A -85,B 0,C 180,E1 -22045.761,E2 -22045.761} C_VEL
LIN {X 0,Y 190.186,Z 550.839,A -85,B 0,C 180,E1 -22049.235,E2 -22049.235} C_VEL
LIN {X 0,Y 190.179,Z 550.739,A -85,B 0,C 180,E1 -22052.117,E2 -22052.117} C_VEL
LIN {X 0,Y 190.168,Z 550.144,A -85,B 0,C 180,E1 -22054.238,E2 -22054.238} C_VEL
LIN {X 0,Y 190.545,Z 547.817,A -85,B 0,C 180,E1 -22058.281,E2 -22058.281} C_VEL
LIN {X 0,Y 190.242,Z 546.493,A -85,B 0,C 180,E1 -22060.01,E2 -22060.01} C_VEL
LIN {X 0,Y 188.198,Z 543.649,A -85,B 0,C 180,E1 -22062.821,E2 -22062.821} C_VEL
LIN {X 0,Y 186.699,Z 540.859,A -85,B 0,C 180,E1 -22065.06,E2 -22065.06} C_VEL
LIN {X 0,Y 186.549,Z 538.528,A -85,B 0,C 180,E1 -22066.73,E2 -22066.73} C_VEL
LIN {X 0,Y 186.803,Z 537.658,A -85,B 0,C 180,E1 -22067.275,E2 -22067.275} C_VEL
LIN {X 0,Y 189.207,Z 531.279,A -85,B 0,C 180,E1 -22070.662,E2 -22070.662} C_VEL
LIN {X 0,Y 191.702,Z 524.779,A -85,B 0,C 180,E1 -22073.377,E2 -22073.377} C_VEL
LIN {X 0,Y 194.068,Z 517.85,A -85,B 0,C 180,E1 -22075.757,E2 -22075.757} C_VEL
LIN {X 0,Y 196.436,Z 510.923,A -85,B 0,C 180,E1 -22077.716,E2 -22077.716} C_VEL
LIN {X 0,Y 197.384,Z 507.073,A -85,B 0,C 180,E1 -22078.729,E2 -22078.729} C_VEL
LIN {X 0,Y 197.673,Z 496.384,A -85,B 0,C 180,E1 -22081.427,E2 -22081.427} C_VEL
LIN {X 0,Y 197.187,Z 486.623,A -85,B 0,C 180,E1 -22083.591,E2 -22083.591} C_VEL
LIN {X 0,Y 195.817,Z 476.909,A -85,B 0,C 180,E1 -22085.599,E2 -22085.599} C_VEL
LIN {X 0,Y 193.738,Z 467.032,A -85,B 0,C 180,E1 -22087.508,E2 -22087.508} C_VEL
LIN {X 0,Y 190.574,Z 456.664,A -85,B 0,C 180,E1 -22089.474,E2 -22089.474} C_VEL
LIN {X 0,Y 187.914,Z 449.497,A -85,B 0,C 180,E1 -22090.842,E2 -22090.842} C_VEL
LIN {X 0,Y 186.519,Z 446.231,A -85,B 0,C 180,E1 -22091.437,E2 -22091.437} C_VEL
LIN {X 0,Y 186.395,Z 445.279,A -85,B 0,C 180,E1 -22091.587,E2 -22091.587} C_VEL
LIN {X 0,Y 186.557,Z 443.067,A -85,B 0,C 180,E1 -22095.705,E2 -22095.705} C_VEL
LIN {X 0,Y 186.378,Z 440.99,A -85,B 0,C 180,E1 -22100.129,E2 -22100.129} C_VEL
LIN {X 0,Y 186.033,Z 438.743,A -85,B 0,C 180,E1 -22105.48,E2 -22105.48} C_VEL
LIN {X 0,Y 185.845,Z 436.865,A -85,B 0,C 180,E1 -22110.552,E2 -22110.552} C_VEL
LIN {X 0,Y 185.659,Z 435.278,A -85,B 0,C 180,E1 -22115.391,E2 -22115.391} C_VEL
LIN {X 0,Y 185.595,Z 434.873,A -85,B 0,C 180,E1 -22117.747,E2 -22117.747} C_VEL
LIN {X 0,Y 185.688,Z 434.857,A -85,B 0,C 180,E1 -22122.374,E2 -22122.374} C_VEL
LIN {X 0,Y 185.74,Z 434.849,A -85,B 0,C 180,E1 -22126.877,E2 -22126.877} C_VEL
LIN {X 0,Y 186.026,Z 434.813,A -85,B 0,C 180,E1 -22131.307,E2 -22131.307} C_VEL
LIN {X 0,Y 186.205,Z 434.79,A -85,B 0,C 180,E1 -22137.836,E2 -22137.836} C_VEL
LIN {X 0,Y 186.403,Z 434.745,A -85,B 0,C 180,E1 -22139.999,E2 -22139.999} C_VEL
LIN {X 0,Y 185.921,Z 434.809,A -85,B 0,C 180,E1 -22144.335,E2 -22144.335} C_VEL
LIN {X 0,Y 186.005,Z 434.811,A -85,B 0,C 180,E1 -22148.692,E2 -22148.692} C_VEL
LIN {X 0,Y 185.76,Z 434.845,A -85,B 0,C 180,E1 -22153.119,E2 -22153.119} C_VEL
LIN {X 0,Y 185.671,Z 434.853,A -85,B 0,C 180,E1 -22158.866,E2 -22158.866} C_VEL
LIN {X 0,Y 185.592,Z 434.868,A -85,B 0,C 180,E1 -22162.251,E2 -22162.251} C_VEL
LIN {X 0,Y 185.558,Z 434.87,A -85,B 0,C 180,E1 -22167.031,E2 -22167.031} C_VEL
LIN {X 0,Y 185.575,Z 434.868,A -85,B 0,C 180,E1 -22169.492,E2 -22169.492} C_VEL
LIN {X 0,Y 185.516,Z 434.876,A -85,B 0,C 180,E1 -22174.627,E2 -22174.627} C_VEL
LIN {X 0,Y 185.563,Z 434.871,A -85,B 0,C 180,E1 -22177.313,E2 -22177.313} C_VEL
LIN {X 0,Y 185.578,Z 434.867,A -85,B 0,C 180,E1 -22180.765,E2 -22180.765} C_VEL
LIN {X 0,Y 185.58,Z 434.87,A -85,B 0,C 180,E1 -22186.014,E2 -22186.014} C_VEL
LIN {X 0,Y 185.572,Z 435.02,A -85,B 0,C 180,E1 -22188.104,E2 -22188.104} C_VEL
LIN {X 0,Y 186.488,Z 437.628,A -85,B 0,C 180,E1 -22188.536,E2 -22188.536} C_VEL
LIN {X 0,Y 188.347,Z 440.05,A -85,B 0,C 180,E1 -22189.2,E2 -22189.2} C_VEL
LIN {X 0,Y 193.064,Z 448.401,A -85,B 0,C 180,E1 -22191.189,E2 -22191.189} C_VEL
LIN {X 0,Y 197.921,Z 458.035,A -85,B 0,C 180,E1 -22193.452,E2 -22193.452} C_VEL
LIN {X 0,Y 202.773,Z 470.298,A -85,B 0,C 180,E1 -22196.285,E2 -22196.285} C_VEL
LIN {X 0,Y 205.656,Z 480.296,A -85,B 0,C 180,E1 -22198.684,E2 -22198.684} C_VEL
LIN {X 0,Y 208.528,Z 489.495,A -85,B 0,C 180,E1 -22201.194,E2 -22201.194} C_VEL
LIN {X 0,Y 212.276,Z 497.875,A -85,B 0,C 180,E1 -22203.893,E2 -22203.893} C_VEL
LIN {X 0,Y 216.769,Z 505.098,A -85,B 0,C 180,E1 -22206.586,E2 -22206.586} C_VEL
LIN {X 0,Y 223.048,Z 512.388,A -85,B 0,C 180,E1 -22209.721,E2 -22209.721} C_VEL
LIN {X 0,Y 228.776,Z 517.571,A -85,B 0,C 180,E1 -22212.232,E2 -22212.232} C_VEL
LIN {X 0,Y 236.25,Z 522.984,A -85,B 0,C 180,E1 -22215.191,E2 -22215.191} C_VEL
LIN {X 0,Y 245.128,Z 528.083,A -85,B 0,C 180,E1 -22218.423,E2 -22218.423} C_VEL
LIN {X 0,Y 252.953,Z 531.748,A -85,B 0,C 180,E1 -22221.211,E2 -22221.211} C_VEL
LIN {X 0,Y 255.41,Z 532.802,A -85,B 0,C 180,E1 -22222.128,E2 -22222.128} C_VEL
LIN {X 0,Y 261.228,Z 535.068,A -85,B 0,C 180,E1 -22224.513,E2 -22224.513} C_VEL
LIN {X 0,Y 262.952,Z 535.697,A -85,B 0,C 180,E1 -22225.401,E2 -22225.401} C_VEL
LIN {X 0,Y 265.461,Z 536.627,A -85,B 0,C 180,E1 -22226.965,E2 -22226.965} C_VEL
LIN {X 0,Y 267.658,Z 537.144,A -85,B 0,C 180,E1 -22228.496,E2 -22228.496} C_VEL
LIN {X 0,Y 269.039,Z 537.292,A -85,B 0,C 180,E1 -22230,E2 -22230} C_VEL
LIN {X 0,Y 267.197,Z 537.045,A -85,B 0,C 180,E1 -22231.836,E2 -22231.836} C_VEL
LIN {X 0,Y 265.428,Z 536.627,A -85,B 0,C 180,E1 -22233.036,E2 -22233.036} C_VEL
LIN {X 0,Y 262.914,Z 535.697,A -85,B 0,C 180,E1 -22234.6,E2 -22234.6} C_VEL
LIN {X 0,Y 259.498,Z 534.432,A -85,B 0,C 180,E1 -22236.219,E2 -22236.219} C_VEL
LIN {X 0,Y 255.351,Z 532.76,A -85,B 0,C 180,E1 -22237.91,E2 -22237.91} C_VEL
LIN {X 0,Y 247.806,Z 529.383,A -85,B 0,C 180,E1 -22240.664,E2 -22240.664} C_VEL
LIN {X 0,Y 238.87,Z 524.605,A -85,B 0,C 180,E1 -22243.855,E2 -22243.855} C_VEL
LIN {X 0,Y 231.22,Z 519.478,A -85,B 0,C 180,E1 -22246.778,E2 -22246.778} C_VEL
LIN {X 0,Y 224.101,Z 513.392,A -85,B 0,C 180,E1 -22249.812,E2 -22249.812} C_VEL
LIN {X 0,Y 218,Z 506.701,A -85,B 0,C 180,E1 -22252.759,E2 -22252.759} C_VEL
LIN {X 0,Y 213.067,Z 499.3,A -85,B 0,C 180,E1 -22255.6,E2 -22255.6} C_VEL
LIN {X 0,Y 209.548,Z 492.117,A -85,B 0,C 180,E1 -22258.005,E2 -22258.005} C_VEL
LIN {X 0,Y 206.615,Z 483.84,A -85,B 0,C 180,E1 -22260.393,E2 -22260.393} C_VEL
LIN {X 0,Y 204.251,Z 475.187,A -85,B 0,C 180,E1 -22262.545,E2 -22262.545} C_VEL
LIN {X 0,Y 201.621,Z 467.237,A -85,B 0,C 180,E1 -22264.427,E2 -22264.427} C_VEL
LIN {X 0,Y 197.912,Z 458.08,A -85,B 0,C 180,E1 -22266.544,E2 -22266.544} C_VEL
LIN {X 0,Y 192.924,Z 448.212,A -85,B 0,C 180,E1 -22268.863,E2 -22268.863} C_VEL
LIN {X 0,Y 189.751,Z 442.628,A -85,B 0,C 180,E1 -22270.208,E2 -22270.208} C_VEL
LIN {X 0,Y 187.728,Z 439.149,A -85,B 0,C 180,E1 -22271.038,E2 -22271.038} C_VEL
LIN {X 0,Y 186.116,Z 436.913,A -85,B 0,C 180,E1 -22271.64,E2 -22271.64} C_VEL
LIN {X 0,Y 185.528,Z 434.875,A -85,B 0,C 180,E1 -22271.964,E2 -22271.964} C_VEL
LIN {X 0,Y 185.51,Z 434.878,A -85,B 0,C 180,E1 -22276.039,E2 -22276.039} C_VEL
LIN {X 0,Y 185.494,Z 434.878,A -85,B 0,C 180,E1 -22279.904,E2 -22279.904} C_VEL
LIN {X 0,Y 185.541,Z 434.874,A -85,B 0,C 180,E1 -22282.697,E2 -22282.697} C_VEL
LIN {X 0,Y 185.543,Z 434.874,A -85,B 0,C 180,E1 -22287.976,E2 -22287.976} C_VEL
LIN {X 0,Y 185.58,Z 434.867,A -85,B 0,C 180,E1 -22290.577,E2 -22290.577} C_VEL
LIN {X 0,Y 185.585,Z 434.859,A -85,B 0,C 180,E1 -22295.384,E2 -22295.384} C_VEL
LIN {X 0,Y 185.606,Z 434.858,A -85,B 0,C 180,E1 -22300.076,E2 -22300.076} C_VEL
LIN {X 0,Y 185.699,Z 434.846,A -85,B 0,C 180,E1 -22304.639,E2 -22304.639} C_VEL
LIN {X 0,Y 185.923,Z 434.82,A -85,B 0,C 180,E1 -22309.36,E2 -22309.36} C_VEL
LIN {X 0,Y 185.96,Z 434.821,A -85,B 0,C 180,E1 -22313.491,E2 -22313.491} C_VEL
LIN {X 0,Y 186.207,Z 434.756,A -85,B 0,C 180,E1 -22317.838,E2 -22317.838} C_VEL
LIN {X 0,Y 186.406,Z 434.745,A -85,B 0,C 180,E1 -22320.001,E2 -22320.001} C_VEL
LIN {X 0,Y 185.926,Z 434.824,A -85,B 0,C 180,E1 -22324.337,E2 -22324.337} C_VEL
LIN {X 0,Y 186.029,Z 434.812,A -85,B 0,C 180,E1 -22328.693,E2 -22328.693} C_VEL
LIN {X 0,Y 185.743,Z 434.849,A -85,B 0,C 180,E1 -22333.123,E2 -22333.123} C_VEL
LIN {X 0,Y 185.691,Z 434.855,A -85,B 0,C 180,E1 -22337.626,E2 -22337.626} C_VEL
LIN {X 0,Y 185.598,Z 434.866,A -85,B 0,C 180,E1 -22342.252,E2 -22342.252} C_VEL
LIN {X 0,Y 185.653,Z 435.302,A -85,B 0,C 180,E1 -22344.697,E2 -22344.697} C_VEL
LIN {X 0,Y 185.854,Z 436.905,A -85,B 0,C 180,E1 -22349.572,E2 -22349.572} C_VEL
LIN {X 0,Y 186.036,Z 438.741,A -85,B 0,C 180,E1 -22354.519,E2 -22354.519} C_VEL
LIN {X 0,Y 186.386,Z 440.996,A -85,B 0,C 180,E1 -22359.869,E2 -22359.869} C_VEL
LIN {X 0,Y 186.561,Z 443.089,A -85,B 0,C 180,E1 -22364.295,E2 -22364.295} C_VEL
LIN {X 0,Y 186.401,Z 445.263,A -85,B 0,C 180,E1 -22368.411,E2 -22368.411} C_VEL
LIN {X 0,Y 187.381,Z 448.526,A -85,B 0,C 180,E1 -22368.946,E2 -22368.946} C_VEL
LIN {X 0,Y 188.475,Z 450.664,A -85,B 0,C 180,E1 -22369.409,E2 -22369.409} C_VEL
LIN {X 0,Y 192.214,Z 461.547,A -85,B 0,C 180,E1 -22371.445,E2 -22371.445} C_VEL
LIN {X 0,Y 194.992,Z 472.514,A -85,B 0,C 180,E1 -22373.54,E2 -22373.54} C_VEL
LIN {X 0,Y 196.575,Z 481.427,A -85,B 0,C 180,E1 -22375.318,E2 -22375.318} C_VEL
LIN {X 0,Y 197.474,Z 491.009,A -85,B 0,C 180,E1 -22377.355,E2 -22377.355} C_VEL
LIN {X 0,Y 197.698,Z 500.204,A -85,B 0,C 180,E1 -22379.513,E2 -22379.513} C_VEL
LIN {X 0,Y 197.362,Z 507.069,A -85,B 0,C 180,E1 -22381.267,E2 -22381.267} C_VEL
LIN {X 0,Y 196.459,Z 510.921,A -85,B 0,C 180,E1 -22382.286,E2 -22382.286} C_VEL
LIN {X 0,Y 193.529,Z 519.476,A -85,B 0,C 180,E1 -22384.742,E2 -22384.742} C_VEL
LIN {X 0,Y 190.629,Z 527.863,A -85,B 0,C 180,E1 -22387.822,E2 -22387.822} C_VEL
LIN {X 0,Y 188.453,Z 533.47,A -85,B 0,C 180,E1 -22390.388,E2 -22390.388} C_VEL
LIN {X 0,Y 186.289,Z 538.964,A -85,B 0,C 180,E1 -22393.564,E2 -22393.564} C_VEL
LIN {X 0,Y 184.793,Z 543.296,A -85,B 0,C 180,E1 -22396.809,E2 -22396.809} C_VEL
LIN {X 0,Y 184.07,Z 545.668,A -85,B 0,C 180,E1 -22398.994,E2 -22398.994} C_VEL
LIN {X 0,Y 183.546,Z 547.473,A -85,B 0,C 180,E1 -22401.19,E2 -22401.19} C_VEL
LIN {X 0,Y 183.081,Z 549.932,A -85,B 0,C 180,E1 -22405.596,E2 -22405.596} C_VEL
LIN {X 0,Y 183.075,Z 550.527,A -85,B 0,C 180,E1 -22407.8,E2 -22407.8} C_VEL
LIN {X 0,Y 183.145,Z 550.685,A -85,B 0,C 180,E1 -22410,E2 -22410} C_VEL
LIN {X 0,Y 183.056,Z 550.2,A -85,B 0,C 180,E1 -22413.413,E2 -22413.413} C_VEL
LIN {X 0,Y 183.231,Z 548.868,A -85,B 0,C 180,E1 -22416.607,E2 -22416.607} C_VEL
LIN {X 0,Y 183.547,Z 547.474,A -85,B 0,C 180,E1 -22418.809,E2 -22418.809} C_VEL
LIN {X 0,Y 184.389,Z 544.516,A -85,B 0,C 180,E1 -22422.1,E2 -22422.1} C_VEL
LIN {X 0,Y 185.681,Z 540.519,A -85,B 0,C 180,E1 -22425.363,E2 -22425.363} C_VEL
LIN {X 0,Y 186.803,Z 537.658,A -85,B 0,C 180,E1 -22427.275,E2 -22427.275} C_VEL
LIN {X 0,Y 187.224,Z 535.012,A -85,B 0,C 180,E1 -22428.888,E2 -22428.888} C_VEL
LIN {X 0,Y 186.352,Z 530.17,A -85,B 0,C 180,E1 -22431.531,E2 -22431.531} C_VEL
LIN {X 0,Y 185.679,Z 524.818,A -85,B 0,C 180,E1 -22434.096,E2 -22434.096} C_VEL
LIN {X 0,Y 186.402,Z 521.187,A -85,B 0,C 180,E1 -22435.54,E2 -22435.54} C_VEL
LIN {X 0,Y 189.524,Z 512.631,A -85,B 0,C 180,E1 -22438.215,E2 -22438.215} C_VEL
LIN {X 0,Y 190.646,Z 508.786,A -85,B 0,C 180,E1 -22439.238,E2 -22439.238} C_VEL
LIN {X 0,Y 191.177,Z 501.134,A -85,B 0,C 180,E1 -22441.333,E2 -22441.333} C_VEL
LIN {X 0,Y 191.195,Z 493.746,A -85,B 0,C 180,E1 -22443.174,E2 -22443.174} C_VEL
LIN {X 0,Y 190.551,Z 485.191,A -85,B 0,C 180,E1 -22445.16,E2 -22445.16} C_VEL
LIN {X 0,Y 189.242,Z 476.126,A -85,B 0,C 180,E1 -22447.126,E2 -22447.126} C_VEL
LIN {X 0,Y 187.401,Z 467.58,A -85,B 0,C 180,E1 -22448.905,E2 -22448.905} C_VEL
LIN {X 0,Y 184.162,Z 456.867,A -85,B 0,C 180,E1 -22451.09,E2 -22451.09} C_VEL
LIN {X 0,Y 181.145,Z 449.437,A -85,B 0,C 180,E1 -22452.701,E2 -22452.701} C_VEL
LIN {X 0,Y 179.704,Z 446.29,A -85,B 0,C 180,E1 -22453.36,E2 -22453.36} C_VEL
LIN {X 0,Y 179.479,Z 445.014,A -85,B 0,C 180,E1 -22453.568,E2 -22453.568} C_VEL
LIN {X 0,Y 179.407,Z 442.745,A -85,B 0,C 180,E1 -22458.243,E2 -22458.243} C_VEL
LIN {X 0,Y 179.206,Z 441.279,A -85,B 0,C 180,E1 -22461.659,E2 -22461.659} C_VEL
LIN {X 0,Y 178.945,Z 439.294,A -85,B 0,C 180,E1 -22466.642,E2 -22466.642} C_VEL
LIN {X 0,Y 178.843,Z 438.159,A -85,B 0,C 180,E1 -22469.827,E2 -22469.827} C_VEL
LIN {X 0,Y 178.647,Z 436.572,A -85,B 0,C 180,E1 -22474.796,E2 -22474.796} C_VEL
LIN {X 0,Y 178.549,Z 435.988,A -85,B 0,C 180,E1 -22476.819,E2 -22476.819} C_VEL
LIN {X 0,Y 178.648,Z 435.735,A -85,B 0,C 180,E1 -22481.655,E2 -22481.655} C_VEL
LIN {X 0,Y 178.664,Z 435.731,A -85,B 0,C 180,E1 -22486.347,E2 -22486.347} C_VEL
LIN {X 0,Y 178.975,Z 435.692,A -85,B 0,C 180,E1 -22490.962,E2 -22490.962} C_VEL
LIN {X 0,Y 179.151,Z 435.669,A -85,B 0,C 180,E1 -22497.75,E2 -22497.75} C_VEL
LIN {X 0,Y 179.366,Z 435.62,A -85,B 0,C 180,E1 -22499.999,E2 -22499.999} C_VEL
LIN {X 0,Y 178.869,Z 435.688,A -85,B 0,C 180,E1 -22504.506,E2 -22504.506} C_VEL
LIN {X 0,Y 178.956,Z 435.688,A -85,B 0,C 180,E1 -22509.037,E2 -22509.037} C_VEL
LIN {X 0,Y 178.677,Z 435.725,A -85,B 0,C 180,E1 -22513.649,E2 -22513.649} C_VEL
LIN {X 0,Y 178.619,Z 435.73,A -85,B 0,C 180,E1 -22519.215,E2 -22519.215} C_VEL
LIN {X 0,Y 178.52,Z 435.738,A -85,B 0,C 180,E1 -22525.117,E2 -22525.117} C_VEL
LIN {X 0,Y 178.518,Z 435.749,A -85,B 0,C 180,E1 -22529.993,E2 -22529.993} C_VEL
LIN {X 0,Y 178.48,Z 435.753,A -85,B 0,C 180,E1 -22534.219,E2 -22534.219} C_VEL
LIN {X 0,Y 178.481,Z 435.752,A -85,B 0,C 180,E1 -22539.05,E2 -22539.05} C_VEL
LIN {X 0,Y 178.509,Z 435.749,A -85,B 0,C 180,E1 -22542.011,E2 -22542.011} C_VEL
LIN {X 0,Y 178.536,Z 435.747,A -85,B 0,C 180,E1 -22546.073,E2 -22546.073} C_VEL
LIN {X 0,Y 179.537,Z 438.578,A -85,B 0,C 180,E1 -22546.593,E2 -22546.593} C_VEL
LIN {X 0,Y 181.397,Z 440.972,A -85,B 0,C 180,E1 -22547.326,E2 -22547.326} C_VEL
LIN {X 0,Y 183.307,Z 444.224,A -85,B 0,C 180,E1 -22548.21,E2 -22548.21} C_VEL
LIN {X 0,Y 187.79,Z 452.1,A -85,B 0,C 180,E1 -22550.269,E2 -22550.269} C_VEL
LIN {X 0,Y 192.708,Z 462.538,A -85,B 0,C 180,E1 -22552.917,E2 -22552.917} C_VEL
LIN {X 0,Y 196.402,Z 472.361,A -85,B 0,C 180,E1 -22555.386,E2 -22555.386} C_VEL
LIN {X 0,Y 198.728,Z 480.104,A -85,B 0,C 180,E1 -22557.365,E2 -22557.365} C_VEL
LIN {X 0,Y 201.169,Z 489.422,A -85,B 0,C 180,E1 -22559.953,E2 -22559.953} C_VEL
LIN {X 0,Y 204.058,Z 497.193,A -85,B 0,C 180,E1 -22562.477,E2 -22562.477} C_VEL
LIN {X 0,Y 208.416,Z 505.301,A -85,B 0,C 180,E1 -22565.567,E2 -22565.567} C_VEL
LIN {X 0,Y 212.404,Z 510.667,A -85,B 0,C 180,E1 -22567.886,E2 -22567.886} C_VEL
LIN {X 0,Y 219.297,Z 517.563,A -85,B 0,C 180,E1 -22571.309,E2 -22571.309} C_VEL
LIN {X 0,Y 226.271,Z 522.9,A -85,B 0,C 180,E1 -22574.332,E2 -22574.332} C_VEL
LIN {X 0,Y 233.546,Z 527.248,A -85,B 0,C 180,E1 -22577.152,E2 -22577.152} C_VEL
LIN {X 0,Y 242.376,Z 531.409,A -85,B 0,C 180,E1 -22580.351,E2 -22580.351} C_VEL
LIN {X 0,Y 248.127,Z 533.665,A -85,B 0,C 180,E1 -22582.45,E2 -22582.45} C_VEL
LIN {X 0,Y 254.037,Z 535.652,A -85,B 0,C 180,E1 -22584.83,E2 -22584.83} C_VEL
LIN {X 0,Y 257.795,Z 536.857,A -85,B 0,C 180,E1 -22586.875,E2 -22586.875} C_VEL
LIN {X 0,Y 260.215,Z 537.364,A -85,B 0,C 180,E1 -22588.453,E2 -22588.453} C_VEL
LIN {X 0,Y 261.787,Z 537.504,A -85,B 0,C 180,E1 -22590,E2 -22590} C_VEL
LIN {X 0,Y 260.131,Z 537.354,A -85,B 0,C 180,E1 -22591.588,E2 -22591.588} C_VEL
LIN {X 0,Y 257.763,Z 536.857,A -85,B 0,C 180,E1 -22593.126,E2 -22593.126} C_VEL
LIN {X 0,Y 254.036,Z 535.654,A -85,B 0,C 180,E1 -22595.167,E2 -22595.167} C_VEL
LIN {X 0,Y 248.134,Z 533.649,A -85,B 0,C 180,E1 -22597.564,E2 -22597.564} C_VEL
LIN {X 0,Y 241.272,Z 530.919,A -85,B 0,C 180,E1 -22600.066,E2 -22600.066} C_VEL
LIN {X 0,Y 231.436,Z 526.091,A -85,B 0,C 180,E1 -22603.658,E2 -22603.658} C_VEL
LIN {X 0,Y 223.739,Z 521.12,A -85,B 0,C 180,E1 -22606.741,E2 -22606.741} C_VEL
LIN {X 0,Y 216.747,Z 515.268,A -85,B 0,C 180,E1 -22609.898,E2 -22609.898} C_VEL
LIN {X 0,Y 210.407,Z 508.147,A -85,B 0,C 180,E1 -22613.236,E2 -22613.236} C_VEL
LIN {X 0,Y 205.545,Z 500.293,A -85,B 0,C 180,E1 -22616.391,E2 -22616.391} C_VEL
LIN {X 0,Y 202.115,Z 492.36,A -85,B 0,C 180,E1 -22619.131,E2 -22619.131} C_VEL
LIN {X 0,Y 199.777,Z 484.503,A -85,B 0,C 180,E1 -22621.454,E2 -22621.454} C_VEL
LIN {X 0,Y 197.342,Z 475.197,A -85,B 0,C 180,E1 -22623.877,E2 -22623.877} C_VEL
LIN {X 0,Y 193.962,Z 465.756,A -85,B 0,C 180,E1 -22626.275,E2 -22626.275} C_VEL
LIN {X 0,Y 190.876,Z 458.516,A -85,B 0,C 180,E1 -22628.102,E2 -22628.102} C_VEL
LIN {X 0,Y 185.72,Z 448.26,A -85,B 0,C 180,E1 -22630.701,E2 -22630.701} C_VEL
LIN {X 0,Y 181.387,Z 441.03,A -85,B 0,C 180,E1 -22632.672,E2 -22632.672} C_VEL
LIN {X 0,Y 180.325,Z 439.68,A -85,B 0,C 180,E1 -22633.1,E2 -22633.1} C_VEL
LIN {X 0,Y 178.933,Z 437.392,A -85,B 0,C 180,E1 -22633.703,E2 -22633.703} C_VEL
LIN {X 0,Y 178.511,Z 435.75,A -85,B 0,C 180,E1 -22633.969,E2 -22633.969} C_VEL
LIN {X 0,Y 178.422,Z 435.761,A -85,B 0,C 180,E1 -22638.452,E2 -22638.452} C_VEL
LIN {X 0,Y 178.447,Z 435.756,A -85,B 0,C 180,E1 -22643.791,E2 -22643.791} C_VEL
LIN {X 0,Y 178.489,Z 435.751,A -85,B 0,C 180,E1 -22646.549,E2 -22646.549} C_VEL
LIN {X 0,Y 178.521,Z 435.749,A -85,B 0,C 180,E1 -22650.007,E2 -22650.007} C_VEL
LIN {X 0,Y 178.523,Z 435.738,A -85,B 0,C 180,E1 -22654.884,E2 -22654.884} C_VEL
LIN {X 0,Y 178.622,Z 435.73,A -85,B 0,C 180,E1 -22660.785,E2 -22660.785} C_VEL
LIN {X 0,Y 178.68,Z 435.725,A -85,B 0,C 180,E1 -22666.351,E2 -22666.351} C_VEL
LIN {X 0,Y 178.959,Z 435.687,A -85,B 0,C 180,E1 -22670.963,E2 -22670.963} C_VEL
LIN {X 0,Y 179.153,Z 435.634,A -85,B 0,C 180,E1 -22677.753,E2 -22677.753} C_VEL
LIN {X 0,Y 179.369,Z 435.62,A -85,B 0,C 180,E1 -22680.001,E2 -22680.001} C_VEL
LIN {X 0,Y 178.875,Z 435.702,A -85,B 0,C 180,E1 -22684.508,E2 -22684.508} C_VEL
LIN {X 0,Y 178.978,Z 435.691,A -85,B 0,C 180,E1 -22689.038,E2 -22689.038} C_VEL
LIN {X 0,Y 178.667,Z 435.732,A -85,B 0,C 180,E1 -22693.653,E2 -22693.653} C_VEL
LIN {X 0,Y 178.624,Z 435.735,A -85,B 0,C 180,E1 -22699.217,E2 -22699.217} C_VEL
LIN {X 0,Y 178.551,Z 435.979,A -85,B 0,C 180,E1 -22703.181,E2 -22703.181} C_VEL
LIN {X 0,Y 178.729,Z 437.491,A -85,B 0,C 180,E1 -22708.157,E2 -22708.157} C_VEL
LIN {X 0,Y 178.853,Z 438.345,A -85,B 0,C 180,E1 -22710.721,E2 -22710.721} C_VEL
LIN {X 0,Y 179.046,Z 440.36,A -85,B 0,C 180,E1 -22716.072,E2 -22716.072} C_VEL
LIN {X 0,Y 179.243,Z 441.495,A -85,B 0,C 180,E1 -22718.856,E2 -22718.856} C_VEL
LIN {X 0,Y 179.416,Z 442.821,A -85,B 0,C 180,E1 -22721.905,E2 -22721.905} C_VEL
LIN {X 0,Y 179.466,Z 445.032,A -85,B 0,C 180,E1 -22726.437,E2 -22726.437} C_VEL
LIN {X 0,Y 180.528,Z 448.344,A -85,B 0,C 180,E1 -22727.03,E2 -22727.03} C_VEL
LIN {X 0,Y 181.74,Z 450.663,A -85,B 0,C 180,E1 -22727.593,E2 -22727.593} C_VEL
LIN {X 0,Y 184.854,Z 458.775,A -85,B 0,C 180,E1 -22729.29,E2 -22729.29} C_VEL
LIN {X 0,Y 188.141,Z 470.399,A -85,B 0,C 180,E1 -22731.672,E2 -22731.672} C_VEL
LIN {X 0,Y 190.14,Z 481.84,A -85,B 0,C 180,E1 -22734.093,E2 -22734.093} C_VEL
LIN {X 0,Y 191.077,Z 491.084,A -85,B 0,C 180,E1 -22736.188,E2 -22736.188} C_VEL
LIN {X 0,Y 191.236,Z 499.82,A -85,B 0,C 180,E1 -22738.324,E2 -22738.324} C_VEL
LIN {X 0,Y 190.867,Z 506.848,A -85,B 0,C 180,E1 -22740.192,E2 -22740.192} C_VEL
LIN {X 0,Y 190.175,Z 510.708,A -85,B 0,C 180,E1 -22741.287,E2 -22741.287} C_VEL
LIN {X 0,Y 187.103,Z 519.262,A -85,B 0,C 180,E1 -22743.81,E2 -22743.81} C_VEL
LIN {X 0,Y 184.028,Z 527.692,A -85,B 0,C 180,E1 -22747.003,E2 -22747.003} C_VEL
LIN {X 0,Y 181.734,Z 533.258,A -85,B 0,C 180,E1 -22749.632,E2 -22749.632} C_VEL
LIN {X 0,Y 179.463,Z 538.751,A -85,B 0,C 180,E1 -22752.92,E2 -22752.92} C_VEL
LIN {X 0,Y 177.848,Z 543.083,A -85,B 0,C 180,E1 -22756.284,E2 -22756.284} C_VEL
LIN {X 0,Y 177.067,Z 545.456,A -85,B 0,C 180,E1 -22758.553,E2 -22758.553} C_VEL
LIN {X 0,Y 176.504,Z 547.261,A -85,B 0,C 180,E1 -22760.835,E2 -22760.835} C_VEL
LIN {X 0,Y 176.011,Z 549.721,A -85,B 0,C 180,E1 -22765.419,E2 -22765.419} C_VEL
LIN {X 0,Y 175.973,Z 550.315,A -85,B 0,C 180,E1 -22767.711,E2 -22767.711} C_VEL
LIN {X 0,Y 176.054,Z 550.474,A -85,B 0,C 180,E1 -22770,E2 -22770} C_VEL
LIN {X 0,Y 175.974,Z 550.086,A -85,B 0,C 180,E1 -22773.175,E2 -22773.175} C_VEL
LIN {X 0,Y 176.157,Z 548.656,A -85,B 0,C 180,E1 -22776.874,E2 -22776.874} C_VEL
LIN {X 0,Y 176.505,Z 547.262,A -85,B 0,C 180,E1 -22779.164,E2 -22779.164} C_VEL
LIN {X 0,Y 177.438,Z 544.304,A -85,B 0,C 180,E1 -22782.582,E2 -22782.582} C_VEL
LIN {X 0,Y 178.809,Z 540.307,A -85,B 0,C 180,E1 -22785.969,E2 -22785.969} C_VEL
LIN {X 0,Y 180.932,Z 535.176,A -85,B 0,C 180,E1 -22789.278,E2 -22789.278} C_VEL
LIN {X 0,Y 183.06,Z 529.912,A -85,B 0,C 180,E1 -22791.981,E2 -22791.981} C_VEL
LIN {X 0,Y 184.95,Z 525.185,A -85,B 0,C 180,E1 -22794.017,E2 -22794.017} C_VEL
LIN {X 0,Y 186.402,Z 521.187,A -85,B 0,C 180,E1 -22795.54,E2 -22795.54} C_VEL
LIN {X 0,Y 187.119,Z 517.459,A -85,B 0,C 180,E1 -22796.936,E2 -22796.936} C_VEL
LIN {X 0,Y 186.85,Z 513.648,A -85,B 0,C 180,E1 -22798.339,E2 -22798.339} C_VEL
LIN {X 0,Y 185.207,Z 505.77,A -85,B 0,C 180,E1 -22801.098,E2 -22801.098} C_VEL
LIN {X 0,Y 184.766,Z 499.899,A -85,B 0,C 180,E1 -22802.836,E2 -22802.836} C_VEL
LIN {X 0,Y 184.735,Z 492.274,A -85,B 0,C 180,E1 -22804.795,E2 -22804.795} C_VEL
LIN {X 0,Y 184.101,Z 484.366,A -85,B 0,C 180,E1 -22806.709,E2 -22806.709} C_VEL
LIN {X 0,Y 182.708,Z 475.374,A -85,B 0,C 180,E1 -22808.781,E2 -22808.781} C_VEL
LIN {X 0,Y 180.773,Z 466.757,A -85,B 0,C 180,E1 -22810.702,E2 -22810.702} C_VEL
LIN {X 0,Y 177.939,Z 457.701,A -85,B 0,C 180,E1 -22812.743,E2 -22812.743} C_VEL
LIN {X 0,Y 175.984,Z 453.098,A -85,B 0,C 180,E1 -22813.842,E2 -22813.842} C_VEL
LIN {X 0,Y 174.477,Z 449.52,A -85,B 0,C 180,E1 -22814.72,E2 -22814.72} C_VEL
LIN {X 0,Y 172.857,Z 446.62,A -85,B 0,C 180,E1 -22815.496,E2 -22815.496} C_VEL
LIN {X 0,Y 172.399,Z 444.719,A -85,B 0,C 180,E1 -22815.869,E2 -22815.869} C_VEL
LIN {X 0,Y 172.206,Z 442.564,A -85,B 0,C 180,E1 -22820.841,E2 -22820.841} C_VEL
LIN {X 0,Y 171.991,Z 440.896,A -85,B 0,C 180,E1 -22825.103,E2 -22825.103} C_VEL
LIN {X 0,Y 171.751,Z 438.951,A -85,B 0,C 180,E1 -22830.59,E2 -22830.59} C_VEL
LIN {X 0,Y 171.557,Z 437.384,A -85,B 0,C 180,E1 -22835.815,E2 -22835.815} C_VEL
LIN {X 0,Y 171.474,Z 436.706,A -85,B 0,C 180,E1 -22838.353,E2 -22838.353} C_VEL
LIN {X 0,Y 171.578,Z 436.616,A -85,B 0,C 180,E1 -22840.87,E2 -22840.87} C_VEL
LIN {X 0,Y 171.58,Z 436.612,A -85,B 0,C 180,E1 -22845.772,E2 -22845.772} C_VEL
LIN {X 0,Y 171.902,Z 436.574,A -85,B 0,C 180,E1 -22850.587,E2 -22850.587} C_VEL
LIN {X 0,Y 171.822,Z 436.582,A -85,B 0,C 180,E1 -22855.306,E2 -22855.306} C_VEL
LIN {X 0,Y 172.329,Z 436.495,A -85,B 0,C 180,E1 -22859.999,E2 -22859.999} C_VEL
LIN {X 0,Y 171.818,Z 436.567,A -85,B 0,C 180,E1 -22864.691,E2 -22864.691} C_VEL
LIN {X 0,Y 171.885,Z 436.566,A -85,B 0,C 180,E1 -22869.412,E2 -22869.412} C_VEL
LIN {X 0,Y 171.589,Z 436.604,A -85,B 0,C 180,E1 -22874.225,E2 -22874.225} C_VEL
LIN {X 0,Y 171.54,Z 436.61,A -85,B 0,C 180,E1 -22879.561,E2 -22879.561} C_VEL
LIN {X 0,Y 171.458,Z 436.619,A -85,B 0,C 180,E1 -22885.611,E2 -22885.611} C_VEL
LIN {X 0,Y 171.437,Z 436.629,A -85,B 0,C 180,E1 -22890.586,E2 -22890.586} C_VEL
LIN {X 0,Y 171.403,Z 436.635,A -85,B 0,C 180,E1 -22895.031,E2 -22895.031} C_VEL
LIN {X 0,Y 171.434,Z 436.63,A -85,B 0,C 180,E1 -22898.841,E2 -22898.841} C_VEL
LIN {X 0,Y 171.447,Z 436.81,A -85,B 0,C 180,E1 -22903.81,E2 -22903.81} C_VEL
LIN {X 0,Y 172.488,Z 439.532,A -85,B 0,C 180,E1 -22904.388,E2 -22904.388} C_VEL
LIN {X 0,Y 174.577,Z 441.991,A -85,B 0,C 180,E1 -22905.297,E2 -22905.297} C_VEL
LIN {X 0,Y 176.376,Z 445.135,A -85,B 0,C 180,E1 -22906.236,E2 -22906.236} C_VEL
LIN {X 0,Y 180.893,Z 452.787,A -85,B 0,C 180,E1 -22908.489,E2 -22908.489} C_VEL
LIN {X 0,Y 185.654,Z 462.756,A -85,B 0,C 180,E1 -22911.245,E2 -22911.245} C_VEL
LIN {X 0,Y 189.324,Z 472.342,A -85,B 0,C 180,E1 -22913.84,E2 -22913.84} C_VEL
LIN {X 0,Y 192.036,Z 480.996,A -85,B 0,C 180,E1 -22916.234,E2 -22916.234} C_VEL
LIN {X 0,Y 194.102,Z 489.715,A -85,B 0,C 180,E1 -22918.754,E2 -22918.754} C_VEL
LIN {X 0,Y 196.904,Z 498.479,A -85,B 0,C 180,E1 -22921.711,E2 -22921.711} C_VEL
LIN {X 0,Y 200.437,Z 505.665,A -85,B 0,C 180,E1 -22924.565,E2 -22924.565} C_VEL
LIN {X 0,Y 205.118,Z 512.493,A -85,B 0,C 180,E1 -22927.681,E2 -22927.681} C_VEL
LIN {X 0,Y 210.271,Z 517.841,A -85,B 0,C 180,E1 -22930.475,E2 -22930.475} C_VEL
LIN {X 0,Y 216.635,Z 522.961,A -85,B 0,C 180,E1 -22933.496,E2 -22933.496} C_VEL
LIN {X 0,Y 223.983,Z 527.506,A -85,B 0,C 180,E1 -22936.576,E2 -22936.576} C_VEL
LIN {X 0,Y 231.783,Z 531.201,A -85,B 0,C 180,E1 -22939.518,E2 -22939.518} C_VEL
LIN {X 0,Y 237.197,Z 533.308,A -85,B 0,C 180,E1 -22941.481,E2 -22941.481} C_VEL
LIN {X 0,Y 242.254,Z 534.951,A -85,B 0,C 180,E1 -22943.337,E2 -22943.337} C_VEL
LIN {X 0,Y 246.843,Z 536.24,A -85,B 0,C 180,E1 -22945.196,E2 -22945.196} C_VEL
LIN {X 0,Y 250.016,Z 537.09,A -85,B 0,C 180,E1 -22946.778,E2 -22946.778} C_VEL
LIN {X 0,Y 253.072,Z 537.652,A -85,B 0,C 180,E1 -22948.67,E2 -22948.67} C_VEL
LIN {X 0,Y 254.485,Z 537.717,A -85,B 0,C 180,E1 -22950,E2 -22950} C_VEL
LIN {X 0,Y 252.618,Z 537.589,A -85,B 0,C 180,E1 -22951.595,E2 -22951.595} C_VEL
LIN {X 0,Y 249.993,Z 537.09,A -85,B 0,C 180,E1 -22953.223,E2 -22953.223} C_VEL
LIN {X 0,Y 246.594,Z 536.179,A -85,B 0,C 180,E1 -22954.905,E2 -22954.905} C_VEL
LIN {X 0,Y 240.852,Z 534.476,A -85,B 0,C 180,E1 -22957.21,E2 -22957.21} C_VEL
LIN {X 0,Y 235.029,Z 532.463,A -85,B 0,C 180,E1 -22959.331,E2 -22959.331} C_VEL
LIN {X 0,Y 226.261,Z 528.649,A -85,B 0,C 180,E1 -22962.558,E2 -22962.558} C_VEL
LIN {X 0,Y 218.844,Z 524.431,A -85,B 0,C 180,E1 -22965.548,E2 -22965.548} C_VEL
LIN {X 0,Y 211.627,Z 519.05,A -85,B 0,C 180,E1 -22968.839,E2 -22968.839} C_VEL
LIN {X 0,Y 205.499,Z 512.932,A -85,B 0,C 180,E1 -22972.098,E2 -22972.098} C_VEL
LIN {X 0,Y 201.299,Z 507.117,A -85,B 0,C 180,E1 -22974.807,E2 -22974.807} C_VEL
LIN {X 0,Y 197.405,Z 499.642,A -85,B 0,C 180,E1 -22977.849,E2 -22977.849} C_VEL
LIN {X 0,Y 194.871,Z 492.6,A -85,B 0,C 180,E1 -22980.325,E2 -22980.325} C_VEL
LIN {X 0,Y 193.056,Z 485.255,A -85,B 0,C 180,E1 -22982.561,E2 -22982.561} C_VEL
LIN {X 0,Y 191.32,Z 478.294,A -85,B 0,C 180,E1 -22984.522,E2 -22984.522} C_VEL
LIN {X 0,Y 187.95,Z 468.477,A -85,B 0,C 180,E1 -22987.208,E2 -22987.208} C_VEL
LIN {X 0,Y 184.342,Z 459.822,A -85,B 0,C 180,E1 -22989.565,E2 -22989.565} C_VEL
LIN {X 0,Y 178.845,Z 449.282,A -85,B 0,C 180,E1 -22992.542,E2 -22992.542} C_VEL
LIN {X 0,Y 175.978,Z 444.712,A -85,B 0,C 180,E1 -22993.938,E2 -22993.938} C_VEL
LIN {X 0,Y 173.97,Z 441.243,A -85,B 0,C 180,E1 -22994.975,E2 -22994.975} C_VEL
LIN {X 0,Y 172.039,Z 438.894,A -85,B 0,C 180,E1 -22995.837,E2 -22995.837} C_VEL
LIN {X 0,Y 171.37,Z 436.639,A -85,B 0,C 180,E1 -22996.3,E2 -22996.3} C_VEL
LIN {X 0,Y 171.412,Z 436.632,A -85,B 0,C 180,E1 -23002.049,E2 -23002.049} C_VEL
LIN {X 0,Y 171.409,Z 436.634,A -85,B 0,C 180,E1 -23005.087,E2 -23005.087} C_VEL
LIN {X 0,Y 171.447,Z 436.628,A -85,B 0,C 180,E1 -23010.536,E2 -23010.536} C_VEL
LIN {X 0,Y 171.451,Z 436.621,A -85,B 0,C 180,E1 -23015.802,E2 -23015.802} C_VEL
LIN {X 0,Y 171.578,Z 436.607,A -85,B 0,C 180,E1 -23020.873,E2 -23020.873} C_VEL
LIN {X 0,Y 171.592,Z 436.603,A -85,B 0,C 180,E1 -23025.776,E2 -23025.776} C_VEL
LIN {X 0,Y 171.888,Z 436.566,A -85,B 0,C 180,E1 -23030.588,E2 -23030.588} C_VEL
LIN {X 0,Y 171.82,Z 436.567,A -85,B 0,C 180,E1 -23035.309,E2 -23035.309} C_VEL
LIN {X 0,Y 172.332,Z 436.495,A -85,B 0,C 180,E1 -23040.001,E2 -23040.001} C_VEL
LIN {X 0,Y 171.825,Z 436.581,A -85,B 0,C 180,E1 -23044.694,E2 -23044.694} C_VEL
LIN {X 0,Y 171.905,Z 436.573,A -85,B 0,C 180,E1 -23049.413,E2 -23049.413} C_VEL
LIN {X 0,Y 171.582,Z 436.613,A -85,B 0,C 180,E1 -23054.228,E2 -23054.228} C_VEL
LIN {X 0,Y 171.546,Z 436.617,A -85,B 0,C 180,E1 -23059.563,E2 -23059.563} C_VEL
LIN {X 0,Y 171.476,Z 436.7,A -85,B 0,C 180,E1 -23061.647,E2 -23061.647} C_VEL
LIN {X 0,Y 171.629,Z 438.129,A -85,B 0,C 180,E1 -23066.773,E2 -23066.773} C_VEL
LIN {X 0,Y 171.829,Z 439.429,A -85,B 0,C 180,E1 -23070.804,E2 -23070.804} C_VEL
LIN {X 0,Y 171.998,Z 441.014,A -85,B 0,C 180,E1 -23075.193,E2 -23075.193} C_VEL
LIN {X 0,Y 172.212,Z 442.567,A -85,B 0,C 180,E1 -23079.159,E2 -23079.159} C_VEL
LIN {X 0,Y 172.409,Z 444.79,A -85,B 0,C 180,E1 -23084.193,E2 -23084.193} C_VEL
LIN {X 0,Y 173.488,Z 448.009,A -85,B 0,C 180,E1 -23084.821,E2 -23084.821} C_VEL
LIN {X 0,Y 174.992,Z 450.491,A -85,B 0,C 180,E1 -23085.553,E2 -23085.553} C_VEL
LIN {X 0,Y 178.521,Z 459.028,A -85,B 0,C 180,E1 -23087.576,E2 -23087.576} C_VEL
LIN {X 0,Y 181.959,Z 471.431,A -85,B 0,C 180,E1 -23090.34,E2 -23090.34} C_VEL
LIN {X 0,Y 183.713,Z 481.197,A -85,B 0,C 180,E1 -23092.544,E2 -23092.544} C_VEL
LIN {X 0,Y 184.696,Z 491.152,A -85,B 0,C 180,E1 -23094.924,E2 -23094.924} C_VEL
LIN {X 0,Y 184.819,Z 499.594,A -85,B 0,C 180,E1 -23097.088,E2 -23097.088} C_VEL
LIN {X 0,Y 184.411,Z 506.625,A -85,B 0,C 180,E1 -23099.037,E2 -23099.037} C_VEL
LIN {X 0,Y 183.871,Z 510.493,A -85,B 0,C 180,E1 -23100.205,E2 -23100.205} C_VEL
LIN {X 0,Y 180.715,Z 519.05,A -85,B 0,C 180,E1 -23102.809,E2 -23102.809} C_VEL
LIN {X 0,Y 177.617,Z 527.177,A -85,B 0,C 180,E1 -23105.96,E2 -23105.96} C_VEL
LIN {X 0,Y 175.043,Z 533.044,A -85,B 0,C 180,E1 -23108.817,E2 -23108.817} C_VEL
LIN {X 0,Y 172.667,Z 538.539,A -85,B 0,C 180,E1 -23112.225,E2 -23112.225} C_VEL
LIN {X 0,Y 170.928,Z 542.871,A -85,B 0,C 180,E1 -23115.717,E2 -23115.717} C_VEL
LIN {X 0,Y 170.09,Z 545.244,A -85,B 0,C 180,E1 -23118.077,E2 -23118.077} C_VEL
LIN {X 0,Y 169.482,Z 547.049,A -85,B 0,C 180,E1 -23120.452,E2 -23120.452} C_VEL
LIN {X 0,Y 168.934,Z 549.509,A -85,B 0,C 180,E1 -23125.227,E2 -23125.227} C_VEL
LIN {X 0,Y 168.87,Z 550.104,A -85,B 0,C 180,E1 -23127.614,E2 -23127.614} C_VEL
LIN {X 0,Y 168.965,Z 550.263,A -85,B 0,C 180,E1 -23129.999,E2 -23129.999} C_VEL
LIN {X 0,Y 168.895,Z 549.971,A -85,B 0,C 180,E1 -23132.921,E2 -23132.921} C_VEL
LIN {X 0,Y 168.934,Z 549.51,A -85,B 0,C 180,E1 -23134.772,E2 -23134.772} C_VEL
LIN {X 0,Y 169.483,Z 547.05,A -85,B 0,C 180,E1 -23139.547,E2 -23139.547} C_VEL
LIN {X 0,Y 170.481,Z 544.092,A -85,B 0,C 180,E1 -23143.104,E2 -23143.104} C_VEL
LIN {X 0,Y 171.963,Z 540.095,A -85,B 0,C 180,E1 -23146.623,E2 -23146.623} C_VEL
LIN {X 0,Y 174.224,Z 534.964,A -85,B 0,C 180,E1 -23150.052,E2 -23150.052} C_VEL
LIN {X 0,Y 176.495,Z 529.701,A -85,B 0,C 180,E1 -23152.844,E2 -23152.844} C_VEL
LIN {X 0,Y 178.607,Z 524.43,A -85,B 0,C 180,E1 -23155.171,E2 -23155.171} C_VEL
LIN {X 0,Y 181.324,Z 517.425,A -85,B 0,C 180,E1 -23157.716,E2 -23157.716} C_VEL
LIN {X 0,Y 183.877,Z 510.497,A -85,B 0,C 180,E1 -23159.792,E2 -23159.792} C_VEL
LIN {X 0,Y 184.649,Z 503.393,A -85,B 0,C 180,E1 -23161.876,E2 -23161.876} C_VEL
LIN {X 0,Y 184.766,Z 499.899,A -85,B 0,C 180,E1 -23162.836,E2 -23162.836} C_VEL
LIN {X 0,Y 184.269,Z 495.669,A -85,B 0,C 180,E1 -23164.106,E2 -23164.106} C_VEL
LIN {X 0,Y 182.78,Z 491.785,A -85,B 0,C 180,E1 -23165.437,E2 -23165.437} C_VEL
LIN {X 0,Y 178.238,Z 482.752,A -85,B 0,C 180,E1 -23168.532,E2 -23168.532} C_VEL
LIN {X 0,Y 176.957,Z 478.216,A -85,B 0,C 180,E1 -23169.73,E2 -23169.73} C_VEL
LIN {X 0,Y 174.582,Z 467.33,A -85,B 0,C 180,E1 -23172.35,E2 -23172.35} C_VEL
LIN {X 0,Y 171.62,Z 458.178,A -85,B 0,C 180,E1 -23174.638,E2 -23174.638} C_VEL
LIN {X 0,Y 169.661,Z 453.858,A -85,B 0,C 180,E1 -23175.805,E2 -23175.805} C_VEL
LIN {X 0,Y 167.663,Z 449.558,A -85,B 0,C 180,E1 -23177.036,E2 -23177.036} C_VEL
LIN {X 0,Y 165.837,Z 446.673,A -85,B 0,C 180,E1 -23177.991,E2 -23177.991} C_VEL
LIN {X 0,Y 165.242,Z 444.419,A -85,B 0,C 180,E1 -23178.486,E2 -23178.486} C_VEL
LIN {X 0,Y 164.993,Z 442.519,A -85,B 0,C 180,E1 -23183.39,E2 -23183.39} C_VEL
LIN {X 0,Y 164.806,Z 440.481,A -85,B 0,C 180,E1 -23189.219,E2 -23189.219} C_VEL
LIN {X 0,Y 164.579,Z 438.789,A -85,B 0,C 180,E1 -23194.719,E2 -23194.719} C_VEL
LIN {X 0,Y 164.483,Z 437.501,A -85,B 0,C 180,E1 -23200.049,E2 -23200.049} C_VEL
LIN {X 0,Y 164.525,Z 437.492,A -85,B 0,C 180,E1 -23205.148,E2 -23205.148} C_VEL
LIN {X 0,Y 164.832,Z 437.454,A -85,B 0,C 180,E1 -23210.179,E2 -23210.179} C_VEL
LIN {X 0,Y 164.858,Z 437.45,A -85,B 0,C 180,E1 -23212.651,E2 -23212.651} C_VEL
LIN {X 0,Y 165.048,Z 437.425,A -85,B 0,C 180,E1 -23217.558,E2 -23217.558} C_VEL
LIN {X 0,Y 165.292,Z 437.37,A -85,B 0,C 180,E1 -23219.999,E2 -23219.999} C_VEL
LIN {X 0,Y 164.767,Z 437.446,A -85,B 0,C 180,E1 -23224.892,E2 -23224.892} C_VEL
LIN {X 0,Y 164.848,Z 437.451,A -85,B 0,C 180,E1 -23227.347,E2 -23227.347} C_VEL
LIN {X 0,Y 164.75,Z 437.46,A -85,B 0,C 180,E1 -23231.15,E2 -23231.15} C_VEL
LIN {X 0,Y 164.482,Z 437.496,A -85,B 0,C 180,E1 -23237.402,E2 -23237.402} C_VEL
LIN {X 0,Y 164.469,Z 437.489,A -85,B 0,C 180,E1 -23239.988,E2 -23239.988} C_VEL
LIN {X 0,Y 164.384,Z 437.502,A -85,B 0,C 180,E1 -23246.129,E2 -23246.129} C_VEL
LIN {X 0,Y 164.371,Z 437.508,A -85,B 0,C 180,E1 -23251.228,E2 -23251.228} C_VEL
LIN {X 0,Y 164.347,Z 437.514,A -85,B 0,C 180,E1 -23256.774,E2 -23256.774} C_VEL
LIN {X 0,Y 164.411,Z 437.669,A -85,B 0,C 180,E1 -23261.239,E2 -23261.239} C_VEL
LIN {X 0,Y 165.324,Z 440.239,A -85,B 0,C 180,E1 -23261.825,E2 -23261.825} C_VEL
LIN {X 0,Y 167.629,Z 443.028,A -85,B 0,C 180,E1 -23262.985,E2 -23262.985} C_VEL
LIN {X 0,Y 169.609,Z 446.331,A -85,B 0,C 180,E1 -23264.117,E2 -23264.117} C_VEL
LIN {X 0,Y 170.491,Z 447.686,A -85,B 0,C 180,E1 -23264.591,E2 -23264.591} C_VEL
LIN {X 0,Y 174.886,Z 455.365,A -85,B 0,C 180,E1 -23267.085,E2 -23267.085} C_VEL
LIN {X 0,Y 179.053,Z 463.949,A -85,B 0,C 180,E1 -23269.703,E2 -23269.703} C_VEL
LIN {X 0,Y 182.388,Z 472.342,A -85,B 0,C 180,E1 -23272.175,E2 -23272.175} C_VEL
LIN {X 0,Y 185.36,Z 481.777,A -85,B 0,C 180,E1 -23274.98,E2 -23274.98} C_VEL
LIN {X 0,Y 187.251,Z 490.297,A -85,B 0,C 180,E1 -23277.573,E2 -23277.573} C_VEL
LIN {X 0,Y 189.453,Z 498.424,A -85,B 0,C 180,E1 -23280.394,E2 -23280.394} C_VEL
LIN {X 0,Y 191.78,Z 504.349,A -85,B 0,C 180,E1 -23282.739,E2 -23282.739} C_VEL
LIN {X 0,Y 196.184,Z 512.058,A -85,B 0,C 180,E1 -23286.308,E2 -23286.308} C_VEL
LIN {X 0,Y 201.373,Z 518.117,A -85,B 0,C 180,E1 -23289.574,E2 -23289.574} C_VEL
LIN {X 0,Y 208.911,Z 524.291,A -85,B 0,C 180,E1 -23293.456,E2 -23293.456} C_VEL
LIN {X 0,Y 216.691,Z 528.938,A -85,B 0,C 180,E1 -23296.878,E2 -23296.878} C_VEL
LIN {X 0,Y 225.093,Z 532.588,A -85,B 0,C 180,E1 -23300.113,E2 -23300.113} C_VEL
LIN {X 0,Y 233.558,Z 535.322,A -85,B 0,C 180,E1 -23303.209,E2 -23303.209} C_VEL
LIN {X 0,Y 239.656,Z 536.822,A -85,B 0,C 180,E1 -23305.591,E2 -23305.591} C_VEL
LIN {X 0,Y 241.961,Z 537.332,A -85,B 0,C 180,E1 -23306.67,E2 -23306.67} C_VEL
LIN {X 0,Y 246.014,Z 537.906,A -85,B 0,C 180,E1 -23308.985,E2 -23308.985} C_VEL
LIN {X 0,Y 247.166,Z 537.931,A -85,B 0,C 180,E1 -23310,E2 -23310} C_VEL
LIN {X 0,Y 246.014,Z 537.907,A -85,B 0,C 180,E1 -23311.015,E2 -23311.015} C_VEL
LIN {X 0,Y 241.95,Z 537.331,A -85,B 0,C 180,E1 -23313.331,E2 -23313.331} C_VEL
LIN {X 0,Y 237.993,Z 536.432,A -85,B 0,C 180,E1 -23315.083,E2 -23315.083} C_VEL
LIN {X 0,Y 233.248,Z 535.222,A -85,B 0,C 180,E1 -23316.923,E2 -23316.923} C_VEL
LIN {X 0,Y 225.109,Z 532.587,A -85,B 0,C 180,E1 -23319.887,E2 -23319.887} C_VEL
LIN {X 0,Y 216.558,Z 528.83,A -85,B 0,C 180,E1 -23323.201,E2 -23323.201} C_VEL
LIN {X 0,Y 208.912,Z 524.289,A -85,B 0,C 180,E1 -23326.546,E2 -23326.546} C_VEL
LIN {X 0,Y 201.374,Z 518.115,A -85,B 0,C 180,E1 -23330.426,E2 -23330.426} C_VEL
LIN {X 0,Y 196.211,Z 512.063,A -85,B 0,C 180,E1 -23333.686,E2 -23333.686} C_VEL
LIN {X 0,Y 191.791,Z 504.482,A -85,B 0,C 180,E1 -23337.21,E2 -23337.21} C_VEL
LIN {X 0,Y 188.357,Z 494.969,A -85,B 0,C 180,E1 -23340.89,E2 -23340.89} C_VEL
LIN {X 0,Y 186.238,Z 485.601,A -85,B 0,C 180,E1 -23343.883,E2 -23343.883} C_VEL
LIN {X 0,Y 184.384,Z 478.496,A -85,B 0,C 180,E1 -23346.027,E2 -23346.027} C_VEL
LIN {X 0,Y 180.871,Z 468.335,A -85,B 0,C 180,E1 -23349.004,E2 -23349.004} C_VEL
LIN {X 0,Y 176.658,Z 458.842,A -85,B 0,C 180,E1 -23351.848,E2 -23351.848} C_VEL
LIN {X 0,Y 171.538,Z 449.583,A -85,B 0,C 180,E1 -23354.824,E2 -23354.824} C_VEL
LIN {X 0,Y 169.707,Z 446.516,A -85,B 0,C 180,E1 -23355.826,E2 -23355.826} C_VEL
LIN {X 0,Y 167.647,Z 443.361,A -85,B 0,C 180,E1 -23356.965,E2 -23356.965} C_VEL
LIN {X 0,Y 167.047,Z 442.256,A -85,B 0,C 180,E1 -23357.325,E2 -23357.325} C_VEL
LIN {X 0,Y 165.209,Z 440.175,A -85,B 0,C 180,E1 -23358.241,E2 -23358.241} C_VEL
LIN {X 0,Y 164.314,Z 437.516,A -85,B 0,C 180,E1 -23358.884,E2 -23358.884} C_VEL
LIN {X 0,Y 164.341,Z 437.513,A -85,B 0,C 180,E1 -23364.343,E2 -23364.343} C_VEL
LIN {X 0,Y 164.389,Z 437.506,A -85,B 0,C 180,E1 -23369.136,E2 -23369.136} C_VEL
LIN {X 0,Y 164.409,Z 437.496,A -85,B 0,C 180,E1 -23374.694,E2 -23374.694} C_VEL
LIN {X 0,Y 164.483,Z 437.488,A -85,B 0,C 180,E1 -23380.052,E2 -23380.052} C_VEL
LIN {X 0,Y 164.534,Z 437.48,A -85,B 0,C 180,E1 -23385.152,E2 -23385.152} C_VEL
LIN {X 0,Y 164.808,Z 437.447,A -85,B 0,C 180,E1 -23390.18,E2 -23390.18} C_VEL
LIN {X 0,Y 164.85,Z 437.45,A -85,B 0,C 180,E1 -23392.653,E2 -23392.653} C_VEL
LIN {X 0,Y 165.049,Z 437.388,A -85,B 0,C 180,E1 -23397.561,E2 -23397.561} C_VEL
LIN {X 0,Y 165.295,Z 437.37,A -85,B 0,C 180,E1 -23400.001,E2 -23400.001} C_VEL
LIN {X 0,Y 164.775,Z 437.459,A -85,B 0,C 180,E1 -23404.895,E2 -23404.895} C_VEL
LIN {X 0,Y 164.861,Z 437.45,A -85,B 0,C 180,E1 -23407.349,E2 -23407.349} C_VEL
LIN {X 0,Y 164.751,Z 437.464,A -85,B 0,C 180,E1 -23411.146,E2 -23411.146} C_VEL
LIN {X 0,Y 164.485,Z 437.497,A -85,B 0,C 180,E1 -23417.404,E2 -23417.404} C_VEL
LIN {X 0,Y 164.475,Z 437.499,A -85,B 0,C 180,E1 -23419.99,E2 -23419.99} C_VEL
LIN {X 0,Y 164.634,Z 439.097,A -85,B 0,C 180,E1 -23426.304,E2 -23426.304} C_VEL
LIN {X 0,Y 164.806,Z 440.726,A -85,B 0,C 180,E1 -23431.474,E2 -23431.474} C_VEL
LIN {X 0,Y 164.997,Z 442.517,A -85,B 0,C 180,E1 -23436.609,E2 -23436.609} C_VEL
LIN {X 0,Y 165.269,Z 444.543,A -85,B 0,C 180,E1 -23441.604,E2 -23441.604} C_VEL
LIN {X 0,Y 166.283,Z 447.645,A -85,B 0,C 180,E1 -23442.26,E2 -23442.26} C_VEL
LIN {X 0,Y 168.193,Z 450.413,A -85,B 0,C 180,E1 -23443.26,E2 -23443.26} C_VEL
LIN {X 0,Y 169.913,Z 454.23,A -85,B 0,C 180,E1 -23444.326,E2 -23444.326} C_VEL
LIN {X 0,Y 172.488,Z 460.494,A -85,B 0,C 180,E1 -23445.966,E2 -23445.966} C_VEL
LIN {X 0,Y 175.118,Z 469.113,A -85,B 0,C 180,E1 -23448.081,E2 -23448.081} C_VEL
LIN {X 0,Y 177.19,Z 479.594,A -85,B 0,C 180,E1 -23450.608,E2 -23450.608} C_VEL
LIN {X 0,Y 178.299,Z 490.172,A -85,B 0,C 180,E1 -23453.276,E2 -23453.276} C_VEL
LIN {X 0,Y 178.428,Z 499.57,A -85,B 0,C 180,E1 -23455.81,E2 -23455.81} C_VEL
LIN {X 0,Y 178.033,Z 506.402,A -85,B 0,C 180,E1 -23457.797,E2 -23457.797} C_VEL
LIN {X 0,Y 177.069,Z 512.203,A -85,B 0,C 180,E1 -23459.598,E2 -23459.598} C_VEL
LIN {X 0,Y 173.181,Z 521.787,A -85,B 0,C 180,E1 -23462.835,E2 -23462.835} C_VEL
LIN {X 0,Y 170.486,Z 528.331,A -85,B 0,C 180,E1 -23465.655,E2 -23465.655} C_VEL
LIN {X 0,Y 168.401,Z 532.832,A -85,B 0,C 180,E1 -23467.938,E2 -23467.938} C_VEL
LIN {X 0,Y 165.903,Z 538.328,A -85,B 0,C 180,E1 -23471.475,E2 -23471.475} C_VEL
LIN {X 0,Y 164.004,Z 542.658,A -85,B 0,C 180,E1 -23475.101,E2 -23475.101} C_VEL
LIN {X 0,Y 163.133,Z 545.032,A -85,B 0,C 180,E1 -23477.56,E2 -23477.56} C_VEL
LIN {X 0,Y 162.456,Z 546.837,A -85,B 0,C 180,E1 -23480.035,E2 -23480.035} C_VEL
LIN {X 0,Y 161.854,Z 549.298,A -85,B 0,C 180,E1 -23485.017,E2 -23485.017} C_VEL
LIN {X 0,Y 161.77,Z 549.953,A -85,B 0,C 180,E1 -23487.766,E2 -23487.766} C_VEL
LIN {X 0,Y 161.864,Z 550.052,A -85,B 0,C 180,E1 -23489.999,E2 -23489.999} C_VEL
LIN {X 0,Y 161.8,Z 549.893,A -85,B 0,C 180,E1 -23492.489,E2 -23492.489} C_VEL
LIN {X 0,Y 161.854,Z 549.298,A -85,B 0,C 180,E1 -23494.981,E2 -23494.981} C_VEL
LIN {X 0,Y 162.457,Z 546.838,A -85,B 0,C 180,E1 -23499.964,E2 -23499.964} C_VEL
LIN {X 0,Y 163.531,Z 543.879,A -85,B 0,C 180,E1 -23503.672,E2 -23503.672} C_VEL
LIN {X 0,Y 165.149,Z 539.883,A -85,B 0,C 180,E1 -23507.33,E2 -23507.33} C_VEL
LIN {X 0,Y 167.547,Z 534.752,A -85,B 0,C 180,E1 -23510.887,E2 -23510.887} C_VEL
LIN {X 0,Y 169.963,Z 529.489,A -85,B 0,C 180,E1 -23513.775,E2 -23513.775} C_VEL
LIN {X 0,Y 172.628,Z 523.167,A -85,B 0,C 180,E1 -23516.604,E2 -23516.604} C_VEL
LIN {X 0,Y 175.058,Z 517.213,A -85,B 0,C 180,E1 -23518.799,E2 -23518.799} C_VEL
LIN {X 0,Y 177.056,Z 512.205,A -85,B 0,C 180,E1 -23520.403,E2 -23520.403} C_VEL
LIN {X 0,Y 177.831,Z 508.344,A -85,B 0,C 180,E1 -23521.576,E2 -23521.576} C_VEL
LIN {X 0,Y 178.408,Z 500.551,A -85,B 0,C 180,E1 -23523.904,E2 -23523.904} C_VEL
LIN {X 0,Y 178.409,Z 492.043,A -85,B 0,C 180,E1 -23526.219,E2 -23526.219} C_VEL
LIN {X 0,Y 177.763,Z 484.237,A -85,B 0,C 180,E1 -23528.224,E2 -23528.224} C_VEL
LIN {X 0,Y 176.957,Z 478.216,A -85,B 0,C 180,E1 -23529.73,E2 -23529.73} C_VEL
LIN {X 0,Y 175.588,Z 473.793,A -85,B 0,C 180,E1 -23530.919,E2 -23530.919} C_VEL
LIN {X 0,Y 173.434,Z 469.993,A -85,B 0,C 180,E1 -23532.248,E2 -23532.248} C_VEL
LIN {X 0,Y 166.413,Z 460.756,A -85,B 0,C 180,E1 -23536.016,E2 -23536.016} C_VEL
LIN {X 0,Y 164.953,Z 458.11,A -85,B 0,C 180,E1 -23536.94,E2 -23536.94} C_VEL
LIN {X 0,Y 163.157,Z 454.3,A -85,B 0,C 180,E1 -23538.111,E2 -23538.111} C_VEL
LIN {X 0,Y 161.386,Z 450.799,A -85,B 0,C 180,E1 -23539.279,E2 -23539.279} C_VEL
LIN {X 0,Y 160.809,Z 449.525,A -85,B 0,C 180,E1 -23539.69,E2 -23539.69} C_VEL
LIN {X 0,Y 158.781,Z 446.638,A -85,B 0,C 180,E1 -23540.874,E2 -23540.874} C_VEL
LIN {X 0,Y 158.01,Z 444.118,A -85,B 0,C 180,E1 -23541.485,E2 -23541.485} C_VEL
LIN {X 0,Y 157.872,Z 442.999,A -85,B 0,C 180,E1 -23544.638,E2 -23544.638} C_VEL
LIN {X 0,Y 157.762,Z 441.956,A -85,B 0,C 180,E1 -23547.821,E2 -23547.821} C_VEL
LIN {X 0,Y 157.597,Z 440.244,A -85,B 0,C 180,E1 -23553.514,E2 -23553.514} C_VEL
LIN {X 0,Y 157.443,Z 438.668,A -85,B 0,C 180,E1 -23559.617,E2 -23559.617} C_VEL
LIN {X 0,Y 157.454,Z 438.373,A -85,B 0,C 180,E1 -23564.464,E2 -23564.464} C_VEL
LIN {X 0,Y 157.747,Z 438.336,A -85,B 0,C 180,E1 -23569.733,E2 -23569.733} C_VEL
LIN {X 0,Y 157.818,Z 438.328,A -85,B 0,C 180,E1 -23572.321,E2 -23572.321} C_VEL
LIN {X 0,Y 158.254,Z 438.245,A -85,B 0,C 180,E1 -23579.999,E2 -23579.999} C_VEL
LIN {X 0,Y 157.805,Z 438.329,A -85,B 0,C 180,E1 -23587.677,E2 -23587.677} C_VEL
LIN {X 0,Y 157.679,Z 438.342,A -85,B 0,C 180,E1 -23591.318,E2 -23591.318} C_VEL
LIN {X 0,Y 157.458,Z 438.363,A -85,B 0,C 180,E1 -23595.532,E2 -23595.532} C_VEL
LIN {X 0,Y 157.365,Z 438.376,A -85,B 0,C 180,E1 -23600.932,E2 -23600.932} C_VEL
LIN {X 0,Y 157.307,Z 438.388,A -85,B 0,C 180,E1 -23606.681,E2 -23606.681} C_VEL
LIN {X 0,Y 157.274,Z 438.395,A -85,B 0,C 180,E1 -23612.426,E2 -23612.426} C_VEL
LIN {X 0,Y 157.291,Z 438.392,A -85,B 0,C 180,E1 -23617.474,E2 -23617.474} C_VEL
LIN {X 0,Y 157.269,Z 438.393,A -85,B 0,C 180,E1 -23618.178,E2 -23618.178} C_VEL
LIN {X 0,Y 158.274,Z 441.223,A -85,B 0,C 180,E1 -23618.95,E2 -23618.95} C_VEL
LIN {X 0,Y 160.682,Z 443.884,A -85,B 0,C 180,E1 -23620.333,E2 -23620.333} C_VEL
LIN {X 0,Y 162.555,Z 447.134,A -85,B 0,C 180,E1 -23621.556,E2 -23621.556} C_VEL
LIN {X 0,Y 163.706,Z 448.756,A -85,B 0,C 180,E1 -23622.23,E2 -23622.23} C_VEL
LIN {X 0,Y 167.643,Z 455.352,A -85,B 0,C 180,E1 -23624.685,E2 -23624.685} C_VEL
LIN {X 0,Y 171.751,Z 463.399,A -85,B 0,C 180,E1 -23627.437,E2 -23627.437} C_VEL
LIN {X 0,Y 175.84,Z 473.462,A -85,B 0,C 180,E1 -23630.7,E2 -23630.7} C_VEL
LIN {X 0,Y 178.419,Z 481.796,A -85,B 0,C 180,E1 -23633.34,E2 -23633.34} C_VEL
LIN {X 0,Y 180.216,Z 489.026,A -85,B 0,C 180,E1 -23635.682,E2 -23635.682} C_VEL
LIN {X 0,Y 181.952,Z 497.572,A -85,B 0,C 180,E1 -23638.664,E2 -23638.664} C_VEL
LIN {X 0,Y 184.079,Z 504.389,A -85,B 0,C 180,E1 -23641.414,E2 -23641.414} C_VEL
LIN {X 0,Y 187.866,Z 511.984,A -85,B 0,C 180,E1 -23645.042,E2 -23645.042} C_VEL
LIN {X 0,Y 192.641,Z 518.389,A -85,B 0,C 180,E1 -23648.604,E2 -23648.604} C_VEL
LIN {X 0,Y 199.119,Z 524.13,A -85,B 0,C 180,E1 -23652.356,E2 -23652.356} C_VEL
LIN {X 0,Y 203.958,Z 527.405,A -85,B 0,C 180,E1 -23654.754,E2 -23654.754} C_VEL
LIN {X 0,Y 212.731,Z 531.768,A -85,B 0,C 180,E1 -23658.568,E2 -23658.568} C_VEL
LIN {X 0,Y 220.305,Z 534.462,A -85,B 0,C 180,E1 -23661.461,E2 -23661.461} C_VEL
LIN {X 0,Y 226.275,Z 536.113,A -85,B 0,C 180,E1 -23663.661,E2 -23663.661} C_VEL
LIN {X 0,Y 233.758,Z 537.578,A -85,B 0,C 180,E1 -23666.553,E2 -23666.553} C_VEL
LIN {X 0,Y 237.143,Z 538.048,A -85,B 0,C 180,E1 -23668.302,E2 -23668.302} C_VEL
LIN {X 0,Y 238.964,Z 538.155,A -85,B 0,C 180,E1 -23669.332,E2 -23669.332} C_VEL
LIN {X 0,Y 239.832,Z 538.145,A -85,B 0,C 180,E1 -23670,E2 -23670} C_VEL
LIN {X 0,Y 238.963,Z 538.156,A -85,B 0,C 180,E1 -23670.663,E2 -23670.663} C_VEL
LIN {X 0,Y 237.129,Z 538.048,A -85,B 0,C 180,E1 -23671.699,E2 -23671.699} C_VEL
LIN {X 0,Y 233.761,Z 537.577,A -85,B 0,C 180,E1 -23673.448,E2 -23673.448} C_VEL
LIN {X 0,Y 226.286,Z 536.093,A -85,B 0,C 180,E1 -23676.365,E2 -23676.365} C_VEL
LIN {X 0,Y 218.388,Z 533.874,A -85,B 0,C 180,E1 -23679.26,E2 -23679.26} C_VEL
LIN {X 0,Y 209.128,Z 530.162,A -85,B 0,C 180,E1 -23682.951,E2 -23682.951} C_VEL
LIN {X 0,Y 200.575,Z 525.202,A -85,B 0,C 180,E1 -23686.885,E2 -23686.885} C_VEL
LIN {X 0,Y 194.651,Z 520.377,A -85,B 0,C 180,E1 -23690.162,E2 -23690.162} C_VEL
LIN {X 0,Y 190.605,Z 516.01,A -85,B 0,C 180,E1 -23692.812,E2 -23692.812} C_VEL
LIN {X 0,Y 185.892,Z 508.566,A -85,B 0,C 180,E1 -23696.66,E2 -23696.66} C_VEL
LIN {X 0,Y 182.918,Z 501.034,A -85,B 0,C 180,E1 -23699.966,E2 -23699.966} C_VEL
LIN {X 0,Y 181.33,Z 494.92,A -85,B 0,C 180,E1 -23702.311,E2 -23702.311} C_VEL
LIN {X 0,Y 179.589,Z 486.204,A -85,B 0,C 180,E1 -23705.225,E2 -23705.225} C_VEL
LIN {X 0,Y 177.205,Z 477.661,A -85,B 0,C 180,E1 -23707.981,E2 -23707.981} C_VEL
LIN {X 0,Y 174.066,Z 468.826,A -85,B 0,C 180,E1 -23710.798,E2 -23710.798} C_VEL
LIN {X 0,Y 170.102,Z 460.115,A -85,B 0,C 180,E1 -23713.696,E2 -23713.696} C_VEL
LIN {X 0,Y 166.066,Z 452.555,A -85,B 0,C 180,E1 -23716.357,E2 -23716.357} C_VEL
LIN {X 0,Y 163.368,Z 448.215,A -85,B 0,C 180,E1 -23717.974,E2 -23717.974} C_VEL
LIN {X 0,Y 161.03,Z 444.924,A -85,B 0,C 180,E1 -23719.374,E2 -23719.374} C_VEL
LIN {X 0,Y 160.249,Z 443.35,A -85,B 0,C 180,E1 -23719.927,E2 -23719.927} C_VEL
LIN {X 0,Y 158.147,Z 441.065,A -85,B 0,C 180,E1 -23721.131,E2 -23721.131} C_VEL
LIN {X 0,Y 157.224,Z 438.399,A -85,B 0,C 180,E1 -23721.891,E2 -23721.891} C_VEL
LIN {X 0,Y 157.289,Z 438.392,A -85,B 0,C 180,E1 -23724.49,E2 -23724.49} C_VEL
LIN {X 0,Y 157.293,Z 438.392,A -85,B 0,C 180,E1 -23728.096,E2 -23728.096} C_VEL
LIN {X 0,Y 157.316,Z 438.385,A -85,B 0,C 180,E1 -23733.467,E2 -23733.467} C_VEL
LIN {X 0,Y 157.392,Z 438.371,A -85,B 0,C 180,E1 -23739.669,E2 -23739.669} C_VEL
LIN {X 0,Y 157.461,Z 438.362,A -85,B 0,C 180,E1 -23744.468,E2 -23744.468} C_VEL
LIN {X 0,Y 157.734,Z 438.328,A -85,B 0,C 180,E1 -23749.735,E2 -23749.735} C_VEL
LIN {X 0,Y 157.808,Z 438.328,A -85,B 0,C 180,E1 -23752.323,E2 -23752.323} C_VEL
LIN {X 0,Y 158.257,Z 438.244,A -85,B 0,C 180,E1 -23760.001,E2 -23760.001} C_VEL
LIN {X 0,Y 157.821,Z 438.328,A -85,B 0,C 180,E1 -23767.679,E2 -23767.679} C_VEL
LIN {X 0,Y 157.68,Z 438.345,A -85,B 0,C 180,E1 -23771.315,E2 -23771.315} C_VEL
LIN {X 0,Y 157.457,Z 438.374,A -85,B 0,C 180,E1 -23775.535,E2 -23775.535} C_VEL
LIN {X 0,Y 157.446,Z 438.663,A -85,B 0,C 180,E1 -23780.383,E2 -23780.383} C_VEL
LIN {X 0,Y 157.623,Z 440.237,A -85,B 0,C 180,E1 -23786.481,E2 -23786.481} C_VEL
LIN {X 0,Y 157.765,Z 441.999,A -85,B 0,C 180,E1 -23792.316,E2 -23792.316} C_VEL
LIN {X 0,Y 157.959,Z 443.523,A -85,B 0,C 180,E1 -23796.787,E2 -23796.787} C_VEL
LIN {X 0,Y 158.056,Z 444.262,A -85,B 0,C 180,E1 -23798.571,E2 -23798.571} C_VEL
LIN {X 0,Y 159.016,Z 447.071,A -85,B 0,C 180,E1 -23799.27,E2 -23799.27} C_VEL
LIN {X 0,Y 161.276,Z 450.429,A -85,B 0,C 180,E1 -23800.626,E2 -23800.626} C_VEL
LIN {X 0,Y 162.929,Z 453.941,A -85,B 0,C 180,E1 -23801.753,E2 -23801.753} C_VEL
LIN {X 0,Y 164.139,Z 456.217,A -85,B 0,C 180,E1 -23802.511,E2 -23802.511} C_VEL
LIN {X 0,Y 167.148,Z 463.542,A -85,B 0,C 180,E1 -23804.71,E2 -23804.71} C_VEL
LIN {X 0,Y 169.164,Z 470.45,A -85,B 0,C 180,E1 -23806.551,E2 -23806.551} C_VEL
LIN {X 0,Y 171.209,Z 481.349,A -85,B 0,C 180,E1 -23809.412,E2 -23809.412} C_VEL
LIN {X 0,Y 172.001,Z 489.936,A -85,B 0,C 180,E1 -23811.694,E2 -23811.694} C_VEL
LIN {X 0,Y 172.175,Z 498.35,A -85,B 0,C 180,E1 -23814.073,E2 -23814.073} C_VEL
LIN {X 0,Y 171.737,Z 506.179,A -85,B 0,C 180,E1 -23816.464,E2 -23816.464} C_VEL
LIN {X 0,Y 170.873,Z 511.987,A -85,B 0,C 180,E1 -23818.372,E2 -23818.372} C_VEL
LIN {X 0,Y 166.863,Z 521.575,A -85,B 0,C 180,E1 -23821.717,E2 -23821.717} C_VEL
LIN {X 0,Y 164.015,Z 528.119,A -85,B 0,C 180,E1 -23824.628,E2 -23824.628} C_VEL
LIN {X 0,Y 161.816,Z 532.62,A -85,B 0,C 180,E1 -23826.99,E2 -23826.99} C_VEL
LIN {X 0,Y 159.174,Z 538.116,A -85,B 0,C 180,E1 -23830.661,E2 -23830.661} C_VEL
LIN {X 0,Y 157.104,Z 542.445,A -85,B 0,C 180,E1 -23834.43,E2 -23834.43} C_VEL
LIN {X 0,Y 156.177,Z 544.82,A -85,B 0,C 180,E1 -23836.997,E2 -23836.997} C_VEL
LIN {X 0,Y 155.453,Z 546.625,A -85,B 0,C 180,E1 -23839.581,E2 -23839.581} C_VEL
LIN {X 0,Y 154.76,Z 549.086,A -85,B 0,C 180,E1 -23844.788,E2 -23844.788} C_VEL
LIN {X 0,Y 154.687,Z 549.833,A -85,B 0,C 180,E1 -23848.304,E2 -23848.304} C_VEL
LIN {X 0,Y 154.702,Z 549.682,A -85,B 0,C 180,E1 -23852.603,E2 -23852.603} C_VEL
LIN {X 0,Y 154.76,Z 549.086,A -85,B 0,C 180,E1 -23855.21,E2 -23855.21} C_VEL
LIN {X 0,Y 155.453,Z 546.626,A -85,B 0,C 180,E1 -23860.418,E2 -23860.418} C_VEL
LIN {X 0,Y 156.605,Z 543.667,A -85,B 0,C 180,E1 -23864.289,E2 -23864.289} C_VEL
LIN {X 0,Y 158.368,Z 539.671,A -85,B 0,C 180,E1 -23868.097,E2 -23868.097} C_VEL
LIN {X 0,Y 160.892,Z 534.539,A -85,B 0,C 180,E1 -23871.794,E2 -23871.794} C_VEL
LIN {X 0,Y 163.459,Z 529.277,A -85,B 0,C 180,E1 -23874.784,E2 -23874.784} C_VEL
LIN {X 0,Y 165.742,Z 524.147,A -85,B 0,C 180,E1 -23877.209,E2 -23877.209} C_VEL
LIN {X 0,Y 168.161,Z 518.628,A -85,B 0,C 180,E1 -23879.41,E2 -23879.41} C_VEL
LIN {X 0,Y 170.862,Z 511.99,A -85,B 0,C 180,E1 -23881.629,E2 -23881.629} C_VEL
LIN {X 0,Y 171.906,Z 504.089,A -85,B 0,C 180,E1 -23884.203,E2 -23884.203} C_VEL
LIN {X 0,Y 172.214,Z 494.551,A -85,B 0,C 180,E1 -23887.007,E2 -23887.007} C_VEL
LIN {X 0,Y 171.533,Z 484.331,A -85,B 0,C 180,E1 -23889.805,E2 -23889.805} C_VEL
LIN {X 0,Y 170.293,Z 475.91,A -85,B 0,C 180,E1 -23892.022,E2 -23892.022} C_VEL
LIN {X 0,Y 168.256,Z 467.024,A -85,B 0,C 180,E1 -23894.354,E2 -23894.354} C_VEL
LIN {X 0,Y 165.788,Z 459.868,A -85,B 0,C 180,E1 -23896.375,E2 -23896.375} C_VEL
LIN {X 0,Y 164.953,Z 458.11,A -85,B 0,C 180,E1 -23896.94,E2 -23896.94} C_VEL
LIN {X 0,Y 163.355,Z 455.731,A -85,B 0,C 180,E1 -23897.889,E2 -23897.889} C_VEL
LIN {X 0,Y 159.869,Z 453.02,A -85,B 0,C 180,E1 -23899.644,E2 -23899.644} C_VEL
LIN {X 0,Y 153.964,Z 449.559,A -85,B 0,C 180,E1 -23902.738,E2 -23902.738} C_VEL
LIN {X 0,Y 151.755,Z 446.691,A -85,B 0,C 180,E1 -23904.218,E2 -23904.218} C_VEL
LIN {X 0,Y 150.794,Z 443.769,A -85,B 0,C 180,E1 -23905.081,E2 -23905.081} C_VEL
LIN {X 0,Y 150.664,Z 442.535,A -85,B 0,C 180,E1 -23909.127,E2 -23909.127} C_VEL
LIN {X 0,Y 150.575,Z 441.585,A -85,B 0,C 180,E1 -23912.472,E2 -23912.472} C_VEL
LIN {X 0,Y 150.396,Z 440.17,A -85,B 0,C 180,E1 -23918.046,E2 -23918.046} C_VEL
LIN {X 0,Y 150.378,Z 439.519,A -85,B 0,C 180,E1 -23920.903,E2 -23920.903} C_VEL
LIN {X 0,Y 150.445,Z 439.246,A -85,B 0,C 180,E1 -23926.491,E2 -23926.491} C_VEL
LIN {X 0,Y 150.661,Z 439.219,A -85,B 0,C 180,E1 -23929.245,E2 -23929.245} C_VEL
LIN {X 0,Y 150.754,Z 439.207,A -85,B 0,C 180,E1 -23931.959,E2 -23931.959} C_VEL
LIN {X 0,Y 151.215,Z 439.12,A -85,B 0,C 180,E1 -23939.999,E2 -23939.999} C_VEL
LIN {X 0,Y 150.741,Z 439.206,A -85,B 0,C 180,E1 -23948.039,E2 -23948.039} C_VEL
LIN {X 0,Y 150.61,Z 439.223,A -85,B 0,C 180,E1 -23951.504,E2 -23951.504} C_VEL
LIN {X 0,Y 150.364,Z 439.25,A -85,B 0,C 180,E1 -23956.285,E2 -23956.285} C_VEL
LIN {X 0,Y 150.347,Z 439.249,A -85,B 0,C 180,E1 -23960.791,E2 -23960.791} C_VEL
LIN {X 0,Y 150.238,Z 439.271,A -85,B 0,C 180,E1 -23967.28,E2 -23967.28} C_VEL
LIN {X 0,Y 150.214,Z 439.274,A -85,B 0,C 180,E1 -23972.634,E2 -23972.634} C_VEL
LIN {X 0,Y 150.215,Z 439.274,A -85,B 0,C 180,E1 -23974.661,E2 -23974.661} C_VEL
LIN {X 0,Y 151.165,Z 441.975,A -85,B 0,C 180,E1 -23975.53,E2 -23975.53} C_VEL
LIN {X 0,Y 153.151,Z 444.14,A -85,B 0,C 180,E1 -23976.875,E2 -23976.875} C_VEL
LIN {X 0,Y 153.807,Z 444.908,A -85,B 0,C 180,E1 -23977.324,E2 -23977.324} C_VEL
LIN {X 0,Y 155.423,Z 447.852,A -85,B 0,C 180,E1 -23978.555,E2 -23978.555} C_VEL
LIN {X 0,Y 156.961,Z 449.743,A -85,B 0,C 180,E1 -23979.541,E2 -23979.541} C_VEL
LIN {X 0,Y 161.907,Z 458.102,A -85,B 0,C 180,E1 -23983.044,E2 -23983.044} C_VEL
LIN {X 0,Y 165.892,Z 466.079,A -85,B 0,C 180,E1 -23986.069,E2 -23986.069} C_VEL
LIN {X 0,Y 168.775,Z 473.094,A -85,B 0,C 180,E1 -23988.549,E2 -23988.549} C_VEL
LIN {X 0,Y 171.561,Z 481.663,A -85,B 0,C 180,E1 -23991.506,E2 -23991.506} C_VEL
LIN {X 0,Y 173.718,Z 490.326,A -85,B 0,C 180,E1 -23994.547,E2 -23994.547} C_VEL
LIN {X 0,Y 175.297,Z 499.312,A -85,B 0,C 180,E1 -23997.876,E2 -23997.876} C_VEL
LIN {X 0,Y 177.158,Z 506.059,A -85,B 0,C 180,E1 -24000.778,E2 -24000.778} C_VEL
LIN {X 0,Y 179.939,Z 512.4,A -85,B 0,C 180,E1 -24003.936,E2 -24003.936} C_VEL
LIN {X 0,Y 184.164,Z 518.655,A -85,B 0,C 180,E1 -24007.567,E2 -24007.567} C_VEL
LIN {X 0,Y 189.566,Z 523.984,A -85,B 0,C 180,E1 -24011.171,E2 -24011.171} C_VEL
LIN {X 0,Y 196.502,Z 528.74,A -85,B 0,C 180,E1 -24014.938,E2 -24014.938} C_VEL
LIN {X 0,Y 203.205,Z 532.052,A -85,B 0,C 180,E1 -24018.024,E2 -24018.024} C_VEL
LIN {X 0,Y 212.958,Z 535.356,A -85,B 0,C 180,E1 -24021.903,E2 -24021.903} C_VEL
LIN {X 0,Y 219.967,Z 536.964,A -85,B 0,C 180,E1 -24024.5,E2 -24024.5} C_VEL
LIN {X 0,Y 225.311,Z 537.862,A -85,B 0,C 180,E1 -24026.501,E2 -24026.501} C_VEL
LIN {X 0,Y 229.152,Z 538.285,A -85,B 0,C 180,E1 -24028.243,E2 -24028.243} C_VEL
LIN {X 0,Y 232.394,Z 538.362,A -85,B 0,C 180,E1 -24030,E2 -24030} C_VEL
LIN {X 0,Y 229.146,Z 538.285,A -85,B 0,C 180,E1 -24031.758,E2 -24031.758} C_VEL
LIN {X 0,Y 225.108,Z 537.835,A -85,B 0,C 180,E1 -24033.58,E2 -24033.58} C_VEL
LIN {X 0,Y 219.013,Z 536.774,A -85,B 0,C 180,E1 -24035.872,E2 -24035.872} C_VEL
LIN {X 0,Y 212.962,Z 535.35,A -85,B 0,C 180,E1 -24038.103,E2 -24038.103} C_VEL
LIN {X 0,Y 203.255,Z 532.049,A -85,B 0,C 180,E1 -24041.974,E2 -24041.974} C_VEL
LIN {X 0,Y 194.311,Z 527.473,A -85,B 0,C 180,E1 -24046.181,E2 -24046.181} C_VEL
LIN {X 0,Y 186.27,Z 521.024,A -85,B 0,C 180,E1 -24050.913,E2 -24050.913} C_VEL
LIN {X 0,Y 181.491,Z 514.993,A -85,B 0,C 180,E1 -24054.621,E2 -24054.621} C_VEL
LIN {X 0,Y 178.528,Z 509.502,A -85,B 0,C 180,E1 -24057.575,E2 -24057.575} C_VEL
LIN {X 0,Y 176.228,Z 503.02,A -85,B 0,C 180,E1 -24060.605,E2 -24060.605} C_VEL
LIN {X 0,Y 174.565,Z 495.247,A -85,B 0,C 180,E1 -24063.7,E2 -24063.7} C_VEL
LIN {X 0,Y 172.815,Z 486.404,A -85,B 0,C 180,E1 -24066.841,E2 -24066.841} C_VEL
LIN {X 0,Y 170.216,Z 477.316,A -85,B 0,C 180,E1 -24069.988,E2 -24069.988} C_VEL
LIN {X 0,Y 167.378,Z 469.555,A -85,B 0,C 180,E1 -24072.71,E2 -24072.71} C_VEL
LIN {X 0,Y 162.776,Z 459.887,A -85,B 0,C 180,E1 -24076.308,E2 -24076.308} C_VEL
LIN {X 0,Y 158.73,Z 452.774,A -85,B 0,C 180,E1 -24079.228,E2 -24079.228} C_VEL
LIN {X 0,Y 156.184,Z 448.779,A -85,B 0,C 180,E1 -24080.954,E2 -24080.954} C_VEL
LIN {X 0,Y 154.108,Z 445.864,A -85,B 0,C 180,E1 -24082.379,E2 -24082.379} C_VEL
LIN {X 0,Y 153.414,Z 444.333,A -85,B 0,C 180,E1 -24082.962,E2 -24082.962} C_VEL
LIN {X 0,Y 151.266,Z 442.154,A -85,B 0,C 180,E1 -24084.395,E2 -24084.395} C_VEL
LIN {X 0,Y 150.258,Z 439.635,A -85,B 0,C 180,E1 -24085.249,E2 -24085.249} C_VEL
LIN {X 0,Y 150.202,Z 439.276,A -85,B 0,C 180,E1 -24085.437,E2 -24085.437} C_VEL
LIN {X 0,Y 150.206,Z 439.273,A -85,B 0,C 180,E1 -24089.026,E2 -24089.026} C_VEL
LIN {X 0,Y 150.24,Z 439.271,A -85,B 0,C 180,E1 -24092.721,E2 -24092.721} C_VEL
LIN {X 0,Y 150.349,Z 439.249,A -85,B 0,C 180,E1 -24099.209,E2 -24099.209} C_VEL
LIN {X 0,Y 150.367,Z 439.249,A -85,B 0,C 180,E1 -24103.715,E2 -24103.715} C_VEL
LIN {X 0,Y 150.657,Z 439.212,A -85,B 0,C 180,E1 -24109.247,E2 -24109.247} C_VEL
LIN {X 0,Y 150.744,Z 439.205,A -85,B 0,C 180,E1 -24111.961,E2 -24111.961} C_VEL
LIN {X 0,Y 151.218,Z 439.119,A -85,B 0,C 180,E1 -24120.001,E2 -24120.001} C_VEL
LIN {X 0,Y 150.757,Z 439.207,A -85,B 0,C 180,E1 -24128.041,E2 -24128.041} C_VEL
LIN {X 0,Y 150.615,Z 439.226,A -85,B 0,C 180,E1 -24131.508,E2 -24131.508} C_VEL
LIN {X 0,Y 150.364,Z 439.255,A -85,B 0,C 180,E1 -24136.288,E2 -24136.288} C_VEL
LIN {X 0,Y 150.407,Z 439.906,A -85,B 0,C 180,E1 -24140.848,E2 -24140.848} C_VEL
LIN {X 0,Y 150.489,Z 440.879,A -85,B 0,C 180,E1 -24144.856,E2 -24144.856} C_VEL
LIN {X 0,Y 150.586,Z 441.665,A -85,B 0,C 180,E1 -24147.823,E2 -24147.823} C_VEL
LIN {X 0,Y 150.737,Z 443.197,A -85,B 0,C 180,E1 -24152.941,E2 -24152.941} C_VEL
LIN {X 0,Y 150.84,Z 444.059,A -85,B 0,C 180,E1 -24155.008,E2 -24155.008} C_VEL
LIN {X 0,Y 152.063,Z 447.286,A -85,B 0,C 180,E1 -24156.005,E2 -24156.005} C_VEL
LIN {X 0,Y 154.302,Z 450.229,A -85,B 0,C 180,E1 -24157.526,E2 -24157.526} C_VEL
LIN {X 0,Y 156.035,Z 453.881,A -85,B 0,C 180,E1 -24158.87,E2 -24158.87} C_VEL
LIN {X 0,Y 157.22,Z 455.837,A -85,B 0,C 180,E1 -24159.674,E2 -24159.674} C_VEL
LIN {X 0,Y 160.961,Z 464.129,A -85,B 0,C 180,E1 -24162.592,E2 -24162.592} C_VEL
LIN {X 0,Y 163.106,Z 470.969,A -85,B 0,C 180,E1 -24164.666,E2 -24164.666} C_VEL
LIN {X 0,Y 164.895,Z 480.382,A -85,B 0,C 180,E1 -24167.325,E2 -24167.325} C_VEL
LIN {X 0,Y 165.848,Z 490.201,A -85,B 0,C 180,E1 -24170.14,E2 -24170.14} C_VEL
LIN {X 0,Y 165.961,Z 499.267,A -85,B 0,C 180,E1 -24172.883,E2 -24172.883} C_VEL
LIN {X 0,Y 165.436,Z 506.365,A -85,B 0,C 180,E1 -24175.162,E2 -24175.162} C_VEL
LIN {X 0,Y 164.15,Z 513.53,A -85,B 0,C 180,E1 -24177.644,E2 -24177.644} C_VEL
LIN {X 0,Y 160.611,Z 521.362,A -85,B 0,C 180,E1 -24180.51,E2 -24180.51} C_VEL
LIN {X 0,Y 157.592,Z 527.906,A -85,B 0,C 180,E1 -24183.515,E2 -24183.515} C_VEL
LIN {X 0,Y 155.291,Z 532.408,A -85,B 0,C 180,E1 -24185.964,E2 -24185.964} C_VEL
LIN {X 0,Y 152.456,Z 537.903,A -85,B 0,C 180,E1 -24189.773,E2 -24189.773} C_VEL
LIN {X 0,Y 150.233,Z 542.233,A -85,B 0,C 180,E1 -24193.699,E2 -24193.699} C_VEL
LIN {X 0,Y 149.221,Z 544.607,A -85,B 0,C 180,E1 -24196.379,E2 -24196.379} C_VEL
LIN {X 0,Y 148.441,Z 546.413,A -85,B 0,C 180,E1 -24199.083,E2 -24199.083} C_VEL
LIN {X 0,Y 147.692,Z 548.875,A -85,B 0,C 180,E1 -24204.538,E2 -24204.538} C_VEL
LIN {X 0,Y 147.625,Z 549.627,A -85,B 0,C 180,E1 -24208.772,E2 -24208.772} C_VEL
LIN {X 0,Y 147.614,Z 549.471,A -85,B 0,C 180,E1 -24212.728,E2 -24212.728} C_VEL
LIN {X 0,Y 147.692,Z 548.875,A -85,B 0,C 180,E1 -24215.46,E2 -24215.46} C_VEL
LIN {X 0,Y 148.441,Z 546.413,A -85,B 0,C 180,E1 -24220.916,E2 -24220.916} C_VEL
LIN {X 0,Y 149.703,Z 543.455,A -85,B 0,C 180,E1 -24224.963,E2 -24224.963} C_VEL
LIN {X 0,Y 151.624,Z 539.459,A -85,B 0,C 180,E1 -24228.932,E2 -24228.932} C_VEL
LIN {X 0,Y 154.272,Z 534.326,A -85,B 0,C 180,E1 -24232.781,E2 -24232.781} C_VEL
LIN {X 0,Y 157.016,Z 529.065,A -85,B 0,C 180,E1 -24235.874,E2 -24235.874} C_VEL
LIN {X 0,Y 159.961,Z 522.741,A -85,B 0,C 180,E1 -24238.9,E2 -24238.9} C_VEL
LIN {X 0,Y 162.711,Z 516.789,A -85,B 0,C 180,E1 -24241.218,E2 -24241.218} C_VEL
LIN {X 0,Y 164.652,Z 511.772,A -85,B 0,C 180,E1 -24242.97,E2 -24242.97} C_VEL
LIN {X 0,Y 165.757,Z 502.673,A -85,B 0,C 180,E1 -24246.048,E2 -24246.048} C_VEL
LIN {X 0,Y 165.992,Z 494.314,A -85,B 0,C 180,E1 -24248.645,E2 -24248.645} C_VEL
LIN {X 0,Y 165.376,Z 484.543,A -85,B 0,C 180,E1 -24251.495,E2 -24251.495} C_VEL
LIN {X 0,Y 164.239,Z 476.392,A -85,B 0,C 180,E1 -24253.803,E2 -24253.803} C_VEL
LIN {X 0,Y 162.36,Z 468.265,A -85,B 0,C 180,E1 -24256.163,E2 -24256.163} C_VEL
LIN {X 0,Y 159.499,Z 460.536,A -85,B 0,C 180,E1 -24258.626,E2 -24258.626} C_VEL
LIN {X 0,Y 157.128,Z 455.581,A -85,B 0,C 180,E1 -24260.402,E2 -24260.402} C_VEL
LIN {X 0,Y 154.536,Z 450.916,A -85,B 0,C 180,E1 -24262.259,E2 -24262.259} C_VEL
LIN {X 0,Y 153.964,Z 449.559,A -85,B 0,C 180,E1 -24262.738,E2 -24262.738} C_VEL
LIN {X 0,Y 150.052,Z 446.599,A -85,B 0,C 180,E1 -24265.235,E2 -24265.235} C_VEL
LIN {X 0,Y 144.662,Z 443.784,A -85,B 0,C 180,E1 -24268.636,E2 -24268.636} C_VEL
LIN {X 0,Y 143.603,Z 443.398,A -85,B 0,C 180,E1 -24269.509,E2 -24269.509} C_VEL
LIN {X 0,Y 143.462,Z 442.269,A -85,B 0,C 180,E1 -24273.837,E2 -24273.837} C_VEL
LIN {X 0,Y 143.379,Z 440.855,A -85,B 0,C 180,E1 -24279.931,E2 -24279.931} C_VEL
LIN {X 0,Y 143.306,Z 440.264,A -85,B 0,C 180,E1 -24282.886,E2 -24282.886} C_VEL
LIN {X 0,Y 143.592,Z 440.1,A -85,B 0,C 180,E1 -24288.708,E2 -24288.708} C_VEL
LIN {X 0,Y 143.672,Z 440.089,A -85,B 0,C 180,E1 -24291.56,E2 -24291.56} C_VEL
LIN {X 0,Y 144.174,Z 439.995,A -85,B 0,C 180,E1 -24299.998,E2 -24299.998} C_VEL
LIN {X 0,Y 143.662,Z 440.085,A -85,B 0,C 180,E1 -24308.438,E2 -24308.438} C_VEL
LIN {X 0,Y 143.545,Z 440.103,A -85,B 0,C 180,E1 -24311.711,E2 -24311.711} C_VEL
LIN {X 0,Y 143.301,Z 440.135,A -85,B 0,C 180,E1 -24317.112,E2 -24317.112} C_VEL
LIN {X 0,Y 143.272,Z 440.132,A -85,B 0,C 180,E1 -24321.253,E2 -24321.253} C_VEL
LIN {X 0,Y 143.185,Z 440.149,A -85,B 0,C 180,E1 -24327.935,E2 -24327.935} C_VEL
LIN {X 0,Y 143.134,Z 440.155,A -85,B 0,C 180,E1 -24330.419,E2 -24330.419} C_VEL
LIN {X 0,Y 144.059,Z 442.838,A -85,B 0,C 180,E1 -24331.424,E2 -24331.424} C_VEL
LIN {X 0,Y 146.191,Z 445.124,A -85,B 0,C 180,E1 -24333.181,E2 -24333.181} C_VEL
LIN {X 0,Y 146.929,Z 445.823,A -85,B 0,C 180,E1 -24333.75,E2 -24333.75} C_VEL
LIN {X 0,Y 148.657,Z 448.954,A -85,B 0,C 180,E1 -24335.284,E2 -24335.284} C_VEL
LIN {X 0,Y 150.203,Z 450.734,A -85,B 0,C 180,E1 -24336.414,E2 -24336.414} C_VEL
LIN {X 0,Y 152.062,Z 453.876,A -85,B 0,C 180,E1 -24337.929,E2 -24337.929} C_VEL
LIN {X 0,Y 155.724,Z 460.035,A -85,B 0,C 180,E1 -24340.872,E2 -24340.872} C_VEL
LIN {X 0,Y 159.371,Z 467.33,A -85,B 0,C 180,E1 -24343.989,E2 -24343.989} C_VEL
LIN {X 0,Y 162.107,Z 473.818,A -85,B 0,C 180,E1 -24346.554,E2 -24346.554} C_VEL
LIN {X 0,Y 164.723,Z 481.493,A -85,B 0,C 180,E1 -24349.458,E2 -24349.458} C_VEL
LIN {X 0,Y 167.093,Z 490.964,A -85,B 0,C 180,E1 -24353.046,E2 -24353.046} C_VEL
LIN {X 0,Y 168.318,Z 498.843,A -85,B 0,C 180,E1 -24356.097,E2 -24356.097} C_VEL
LIN {X 0,Y 170.009,Z 506.667,A -85,B 0,C 180,E1 -24359.578,E2 -24359.578} C_VEL
LIN {X 0,Y 172.189,Z 512.651,A -85,B 0,C 180,E1 -24362.667,E2 -24362.667} C_VEL
LIN {X 0,Y 176.064,Z 519.222,A -85,B 0,C 180,E1 -24366.646,E2 -24366.646} C_VEL
LIN {X 0,Y 179.895,Z 523.553,A -85,B 0,C 180,E1 -24369.651,E2 -24369.651} C_VEL
LIN {X 0,Y 186.355,Z 528.481,A -85,B 0,C 180,E1 -24373.676,E2 -24373.676} C_VEL
LIN {X 0,Y 194.242,Z 532.536,A -85,B 0,C 180,E1 -24377.657,E2 -24377.657} C_VEL
LIN {X 0,Y 199.769,Z 534.628,A -85,B 0,C 180,E1 -24380.075,E2 -24380.075} C_VEL
LIN {X 0,Y 205.617,Z 536.252,A -85,B 0,C 180,E1 -24382.394,E2 -24382.394} C_VEL
LIN {X 0,Y 211.75,Z 537.439,A -85,B 0,C 180,E1 -24384.673,E2 -24384.673} C_VEL
LIN {X 0,Y 218.152,Z 538.282,A -85,B 0,C 180,E1 -24387.055,E2 -24387.055} C_VEL
LIN {X 0,Y 220.831,Z 538.531,A -85,B 0,C 180,E1 -24388.177,E2 -24388.177} C_VEL
LIN {X 0,Y 224.566,Z 538.591,A -85,B 0,C 180,E1 -24390,E2 -24390} C_VEL
LIN {X 0,Y 220.833,Z 538.531,A -85,B 0,C 180,E1 -24391.824,E2 -24391.824} C_VEL
LIN {X 0,Y 216.094,Z 538.104,A -85,B 0,C 180,E1 -24393.73,E2 -24393.73} C_VEL
LIN {X 0,Y 210.633,Z 537.238,A -85,B 0,C 180,E1 -24395.745,E2 -24395.745} C_VEL
LIN {X 0,Y 204.909,Z 536.062,A -85,B 0,C 180,E1 -24397.886,E2 -24397.886} C_VEL
LIN {X 0,Y 199.273,Z 534.452,A -85,B 0,C 180,E1 -24400.157,E2 -24400.157} C_VEL
LIN {X 0,Y 189.05,Z 530.073,A -85,B 0,C 180,E1 -24404.864,E2 -24404.864} C_VEL
LIN {X 0,Y 181.813,Z 525.203,A -85,B 0,C 180,E1 -24409.049,E2 -24409.049} C_VEL
LIN {X 0,Y 177.581,Z 521.118,A -85,B 0,C 180,E1 -24412.085,E2 -24412.085} C_VEL
LIN {X 0,Y 173.39,Z 515.081,A -85,B 0,C 180,E1 -24415.936,E2 -24415.936} C_VEL
LIN {X 0,Y 170.748,Z 509.116,A -85,B 0,C 180,E1 -24419.22,E2 -24419.22} C_VEL
LIN {X 0,Y 168.74,Z 501.523,A -85,B 0,C 180,E1 -24422.782,E2 -24422.782} C_VEL
LIN {X 0,Y 167.528,Z 493.555,A -85,B 0,C 180,E1 -24425.967,E2 -24425.967} C_VEL
LIN {X 0,Y 166.157,Z 486.881,A -85,B 0,C 180,E1 -24428.514,E2 -24428.514} C_VEL
LIN {X 0,Y 163.91,Z 478.955,A -85,B 0,C 180,E1 -24431.507,E2 -24431.507} C_VEL
LIN {X 0,Y 160.885,Z 470.682,A -85,B 0,C 180,E1 -24434.691,E2 -24434.691} C_VEL
LIN {X 0,Y 156.734,Z 461.918,A -85,B 0,C 180,E1 -24438.328,E2 -24438.328} C_VEL
LIN {X 0,Y 152.926,Z 455.185,A -85,B 0,C 180,E1 -24441.377,E2 -24441.377} C_VEL
LIN {X 0,Y 150.272,Z 451.032,A -85,B 0,C 180,E1 -24443.501,E2 -24443.501} C_VEL
LIN {X 0,Y 149.373,Z 449.774,A -85,B 0,C 180,E1 -24444.186,E2 -24444.186} C_VEL
LIN {X 0,Y 147.379,Z 446.971,A -85,B 0,C 180,E1 -24445.782,E2 -24445.782} C_VEL
LIN {X 0,Y 146.672,Z 445.417,A -85,B 0,C 180,E1 -24446.476,E2 -24446.476} C_VEL
LIN {X 0,Y 144.331,Z 443.232,A -85,B 0,C 180,E1 -24448.335,E2 -24448.335} C_VEL
LIN {X 0,Y 143.264,Z 440.766,A -85,B 0,C 180,E1 -24449.407,E2 -24449.407} C_VEL
LIN {X 0,Y 143.14,Z 440.155,A -85,B 0,C 180,E1 -24449.684,E2 -24449.684} C_VEL
LIN {X 0,Y 143.155,Z 440.146,A -85,B 0,C 180,E1 -24453.78,E2 -24453.78} C_VEL
LIN {X 0,Y 143.306,Z 440.124,A -85,B 0,C 180,E1 -24459.924,E2 -24459.924} C_VEL
LIN {X 0,Y 143.368,Z 440.118,A -85,B 0,C 180,E1 -24465.814,E2 -24465.814} C_VEL
LIN {X 0,Y 143.594,Z 440.094,A -85,B 0,C 180,E1 -24468.712,E2 -24468.712} C_VEL
LIN {X 0,Y 143.664,Z 440.085,A -85,B 0,C 180,E1 -24471.562,E2 -24471.562} C_VEL
LIN {X 0,Y 144.177,Z 439.994,A -85,B 0,C 180,E1 -24480.002,E2 -24480.002} C_VEL
LIN {X 0,Y 143.675,Z 440.088,A -85,B 0,C 180,E1 -24488.44,E2 -24488.44} C_VEL
LIN {X 0,Y 143.549,Z 440.107,A -85,B 0,C 180,E1 -24491.714,E2 -24491.714} C_VEL
LIN {X 0,Y 143.309,Z 440.263,A -85,B 0,C 180,E1 -24497.114,E2 -24497.114} C_VEL
